(* CODESYS project lcls-twincat-motion-v4.0.8.library
   Title: lcls-twincat-motion
   Version: 4.0.8
   Placeholder: lcls-twincat-motion
   Company: SLAC

Project tree, tasks and I/O mapping:
  libraries: LCLS General, * (SLAC); PMPS, * (SLAC - LCLS); Tc2_EtherCAT, * (Beckhoff Automation GmbH); Tc2_Math, * (Beckhoff Automation GmbH); Tc2_MC2, * (Beckhoff Automation GmbH); Tc2_Standard, * (Beckhoff Automation GmbH); Tc2_System, * (Beckhoff Automation GmbH); Tc2_Utilities, * (Beckhoff Automation GmbH); Tc3_JsonXml, * (Beckhoff Automation GmbH); Tc3_Module, * (Beckhoff Automation GmbH); TcUnit, * (www.tcunit.org)
  DUTs/
    Deprecated/
      data type DUT_MotionPneumaticActuator
      data type DUT_MotionStage
      data type DUT_PositionState
      data type EL5042_Status
      data type ENUM_EpicsHomeCmd
      data type ENUM_EpicsInOut
      data type ENUM_EpicsInOut_INT
      data type ENUM_EpicsMotorCmd
      data type ENUM_MotionFFType
      data type ENUM_MotionRequest
      data type ENUM_PnuematicActuatorPositionState
      data type ENUM_StageBrakeMode
      data type ENUM_StageEnableMode
      data type ENUM_StatePMPSStatus
    data type E_EpicsHomeCmd
    data type E_EpicsInOut
    data type E_EpicsMotorCmd
    data type E_LCLSMotionError
    data type E_MotionFFType
    data type E_MotionRequest
    data type E_PnuematicActuatorPositionState
    data type E_StageBrakeMode
    data type E_StageEnableMode
    data type E_StatePMPSStatus
    data type ST_AxisParameterSetExposed
    data type ST_EL5042_Status
    data type ST_MotionPneumaticActuator
    data type ST_MotionStage
    data type ST_PositionState
    data type ST_RenishawAbsEnc
    data type ST_StateEpicsToPlc
    data type ST_StatePlcToEpics
    data type ST_StatePMPSEpicsToPlc
    data type ST_StatePMPSPlcToEpics
  GVLs/
    global variables MOTION_GVL
    global variables MotionConstants
  POUs/
    Deprecated/
      function block FB_EpicsInOut [ST]
      function block FB_PositionStateBase [ST]: Exec, StateHandler
      function block FB_PositionStateBase_WithPMPS [ST]: Exec, PMPSHandler
      function block FB_PositionStateBase_WithPMPS_Test [ST]: Exec, PMPSHandler
      function block FB_PositionStateInOut [ST]
      function block FB_PositionStateInOut_WithPMPS [ST]
      function block FB_PositionStateInOut_WithPMPS_Test [ST]
      function block FB_PositionStateManager [ST]
      function block FB_PositionStatePMPS [ST]: AssertHere, ClearAsserts, HandleBPTM, HandleFFO, HandlePmpsDb
      function block FB_PositionStatePMPS_Base [ST]: AssertHere, ClearAsserts, Exec, GetBeamFromState, GetStateCode, GetStateStruct, HandleBPTM, HandleFFO, HandlePmpsDb
      function block FB_PositionStatePMPS_Test [ST]: HandleBPTM, HandleFFO
      function block FB_StatePTPMove [ST]
    ImplicitChecks/
      function CheckBounds [ST]
      function CheckDivDInt [ST]
      function CheckDivLInt [ST]
      function CheckDivLReal [ST]
      function CheckDivReal [ST]
    Motion/
      Gantry/
        function block FB_GantryAutoCoupling [ST]
        function block FB_GantryDiffVirtualLimitSwitch [ST]
      PMPS/
        function block FB_EncErrorFFO [ST]
        function block FB_MiscStatesErrorFFO [ST]
        function block FB_MotionBPTM [ST]: CheckCount, HandleTimeout, RunBPTM, SetDoneMoving
        function block FB_MotionClearAsserts [ST]
        function block FB_MotionReadPMPSDBND [ST]: BackfillInfo, ReadDatabase, RunFastFaults, SelectLookupKeys
        function block FB_NCErrorFFO [ST]
        function block FB_PerMotorFFOND [ST]: CheckCount, HandleFFO, HandleLoops
        function block FB_PositionStatePMPS1D [ST]
        function block FB_PositionStatePMPS2D [ST]
        function block FB_PositionStatePMPS3D [ST]
        function block FB_PositionStatePMPSND_Core [ST]
        function block FB_Standard_PMPSDB [ST]
        function block FB_StatePMPSEnables [ST]: ApplyEnables, GetBounds, RunFastFaults, SetEnables
        function block FB_StatePMPSEnablesND [ST]: CheckCount, DoLimits, RunFastFaults
      States/
        Examples/
          function block FB_PositionState1D_InOut [ST]
          function block FB_PositionState2D_InOut [ST]
          function block FB_PositionStatePMPS1D_InOut [ST]
          function block FB_PositionStatePMPS2D_InOut [ST]
        Helpers/
          function F_AtPositionState [ST]
          function F_PosOverLowerBound [ST]
          function F_PosUnderUpperBound [ST]
          function F_PosWithinDelta [ST]
          function block FB_RawCountConverter [ST]
        Internals/
          function block FB_PositionStateInternal [ST]
          function block FB_PositionStateInternalND [ST]
          function block FB_PositionStateLock [ST]
        function block FB_PositionState1D [ST]
        function block FB_PositionState2D [ST]
        function block FB_PositionState3D [ST]
        function block FB_PositionStateMove [ST]
        function block FB_PositionStateMoveND [ST]: CheckCount, CombineOutputs, DoStateMoves
        function block FB_PositionStateND_Core [ST]
        function block FB_PositionStateRead [ST]
        function block FB_PositionStateReadND [ST]: CheckCount, CombineOutputs, DoStateReads
        function block FB_StateSetupHelper [ST]
        function block FB_StatesInputHandler [ST]
      Utils/
        function F_MotionErrorCodeLookup [ST]
        function block FB_SetEnables [ST]
      function block FB_EncoderValue [ST]
      function block FB_EncSaveRestore [ST]
      function block FB_LogMotionError [ST]
      function block FB_MotionHoming [ST]
      function block FB_MotionPneumaticActuator [ST]: ACT_IO, ACT_Logger
      function block FB_MotionRequest [ST]
      function block FB_MotionStage [ST]
      function block FB_MotionStageNCParams [ST]
      function block FB_MotionStageSim [ST]
    MotorTesting/
      function block FB_MicroStepCountTest [ST]
  tc_mca_std_lib/
    DUTs/
      data type DUT_AxisStatus_v0_01
    GVLs/
      global variables GVL
    POUs/
      ChangeConfig/
        function block FB_ReadFloatParameter [ST]
        function block FB_ReadParameterInNc_v1_00 [ST]
        function block FB_WriteFloatParameter [ST]
        function block FB_WriteParameterInNc_v1_00 [ST]
      ErrorHandling/
        data type DUT_ErrorState
        data type DUT_TerminalError
        function block FB_ErrorList [ST]
        function block FB_TerminalError [ST]
        global variables GVL_ErrorSystem
        data type ST_ErrorSystem
      Hardware/
        EtherCAT_Terminals/
          Analog_Inputs/
            function block EL3174_0002 [ST]
            function block EL3214 [ST]
            function block EL3255 [ST]
            function block FB_CalculateFrequency_3702_v0_01 [ST]
          Digital_Inputs/
            function block EL1008 [ST]
            function block EL1018 [ST]
            function block EL1808 [ST]
            function block EL1809 [ST]
            function block EL1819 [ST]
            function block FB_EL1252ASM_v1_00 [ST]
          Digital_Outputs/
            External_Types/
              data type dutEL2521_Ctrl
              data type dutEL2521_Status
            function block EL2014 [ST]
            function block EL2252 [ST]
            function block EL2808 [ST]
            function block EL2819 [ST]
          Measuring_Terminals/
            function block EL5002 [ST]
            function block EL5021 [ST]
            function block EL5042 [ST]
            function block EL5101 [ST]
          Motion/
            function block EL7211_v1_00 [ST]
            function block EL9576_v1_00 [ST]
          System/
            function block EL9410 [ST]
            function block EL9505 [ST]
        Other/
          function block EK1200 [ST]
      Motion/
        Homing/
          function block FB_HomeDirect [ST]
          function block FB_HomeFinish [ST]
          function block FB_HomePrepare [ST]
          function block FB_HomeReadNcVelocities [ST]
          function block FB_HomeReadSoftLimEnable [ST]
          function block FB_HomeToSwitch [ST]
          function block FB_HomeVirtual [ST]
          function block FB_HomeWriteNcVelocities [ST]
          function block FB_HomeWriteSoftLimEnable [ST]
        function block FB_DriveVirtual [ST]
        function block FB_NcAxis [ST]
  Tests/
    Helpers/
      data type E_TestStates
      function block FB_CauseNCError [ST]
      function block FB_MotorTestSuite [ST]: SetEnables, SetEnablesPMPS, SetGoodState
      function block FB_PMPSJsonTestHelper [ST]: bitmaskToString
      function block FB_TestHelperSetAndMove [ST]
    function block FB_AtPositionState_Test [ST]: TestAtPositionStateInvalid, TestAtPositionStateJustRight, TestAtPositionStateLeave, TestAtPositionStateTooHigh, TestAtPositionStateTooLow, TestAtPositionStateTweak, TestAtPositionStateWithoutInternal, TestPosOverLowerBoundNo, TestPosOverLowerBoundYes, TestPosUnderUpperBoundNo, TestPosUnderUpperBoundYes, TestPosWithinDeltaJustRight, TestPosWithinDeltaTooHigh, TestPosWithinDeltaTooLow
    function block FB_AxisParameterSetExposed_Test [ST]: TestParameterCopy
    function block FB_MiscStatesErrorFFO_Test [ST]: TestBeamParamsNotOk, TestDebounce, TestTransitionState, TestUnknownState, TestZeroRate, TripUntrip
    function block FB_MotionBPTM_Test [ST]: AssertInPool, SetMotorDone, SetMotorMoving, SetMotorStartup, Test3dMove, TestCount, TestInit, TestNoMove
    function block FB_MotionClearAsserts_Test [ST]: TestBasic
    function block FB_MotionReadPMPSDBND_Test [ST]: TestBackfill, TestDupe, TestHalfFull, TestNonsense, TestSolo, TestTrio
    function block FB_NCErrorFFO_Test [ST]: TestEnc, TestNC
    function block FB_PerMotorFFOND_Test [ST]: TestBlankCount, TestTwoMotorEncError
    function block FB_PositionStateMove_Test [ST]: TestBadStates, TestMove, TestMoveOk
    function block FB_PositionStateMoveND_Test [ST]: ResetGoals, TestMove
    function block FB_PositionStateND_Test [ST]: Test1D, Test2D, Test3D, TestInputDeadlock
    function block FB_PositionStatePMPSND_Test [ST]: AssertMotionLims, Test1D, Test2D, Test3D, TestStartup1D, TestStartup2D, TestStartup3D
    function block FB_PositionStateRead_Test [ST]: Asserts, TestDupe, TestMovingPosition, TestStaticPosition
    function block FB_PositionStateReadND_Test [ST]: DoAssert, DoMove, DoRead, PerMotor, SquareSetup, TestCombos, TestForgot, TestSquare
    function block FB_StatePMPSEnables_Test [ST]: TestAbove, TestAt, TestBelow, TestDisabled, TestInvalid, TestLimits, TestMoveAt, TestMoveTo, TestNotUpdated
    function block FB_StatePMPSEnablesND_Test [ST]: TestCount, TestMaint, TestUnderOverGoals
    function block FB_StateSetupHelper_Test [ST]: TestDefaultOnly, TestManyOverrides, TestNoDefault, TestNormalCase, TestOnlyOnce
    function block FB_TestHelperSetAndMove_Test [ST]: BasicMotion
    function block FB_TestStateInitTiming [ST]: PassiveReinit
    program PRG_TEST [ST]
  Version/
    global variables Global_Version
*)

// DUTs/Deprecated/DUT_MotionPneumaticActuator
{attribute 'obsolete' := 'DUT_MotionPneumaticActuator has been renamed to ST_MotionPneumaticActuator'}
TYPE DUT_MotionPneumaticActuator : ST_MotionPneumaticActuator; END_TYPE

// DUTs/Deprecated/DUT_MotionStage
{attribute 'obsolete' := 'DUT_MotionStage has been renamed to ST_MotionStage'}
TYPE DUT_MotionStage : ST_MotionStage; END_TYPE

// DUTs/Deprecated/DUT_PositionState
{attribute 'obsolete' := 'DUT_PositionState has been renamed to ST_PositionState'}
TYPE DUT_PositionState : ST_PositionState; END_TYPE

// DUTs/Deprecated/EL5042_Status
{attribute 'obsolete' := 'EL5042_Status has been renamed to ST_EL5042_Status'}
TYPE EL5042_Status : ST_EL5042_Status; END_TYPE

// DUTs/Deprecated/ENUM_EpicsHomeCmd
{attribute 'obsolete' := 'Use E_EpicsHomeCmd'}
TYPE ENUM_EpicsHomeCmd : E_EpicsHomeCmd; END_TYPE

// DUTs/Deprecated/ENUM_EpicsInOut
{attribute 'obsolete' := 'Use E_EpicsInOut'}
TYPE ENUM_EpicsInOut : E_EpicsInOut; END_TYPE

// DUTs/Deprecated/ENUM_EpicsInOut_INT
{attribute 'obsolete' := 'Use ENUM_EpicsInOut'}
{attribute 'qualified_only'}
// Example EPICS states enum for use in all versions of the states FBs
// Remove strict attribute for easier handling
TYPE ENUM_EpicsInOut_INT :
(
    UNKNOWN := 0, // UNKNOWN must be in slot 0 or the FB breaks
    OUT := 1, // OUT at slot 1 is a convention
    IN := 2
) INT;
END_TYPE

// DUTs/Deprecated/ENUM_EpicsMotorCmd
{attribute 'obsolete' := 'Use E_EpicsMotorCmd'}
TYPE ENUM_EpicsMotorCmd : E_EpicsMotorCmd; END_TYPE

// DUTs/Deprecated/ENUM_MotionFFType
{attribute 'obsolete' := 'Use E_MotionFFType'}
TYPE ENUM_MotionFFType : E_MotionFFType; END_TYPE

// DUTs/Deprecated/ENUM_MotionRequest
{attribute 'obsolete' := 'Use E_MotionRequest'}
TYPE ENUM_MotionRequest : E_MotionRequest; END_TYPE

// DUTs/Deprecated/ENUM_PnuematicActuatorPositionState
{attribute 'obsolete' := 'Use E_PnuematicActuatorPositionState'}
TYPE ENUM_PnuematicActuatorPositionState : E_PnuematicActuatorPositionState; END_TYPE

// DUTs/Deprecated/ENUM_StageBrakeMode
{attribute 'obsolete' := 'Use E_StageBrakeMode'}
TYPE ENUM_StageBrakeMode : E_StageBrakeMode; END_TYPE

// DUTs/Deprecated/ENUM_StageEnableMode
{attribute 'obsolete' := 'Use E_StageEnableMode'}
TYPE ENUM_StageEnableMode : E_StageEnableMode; END_TYPE

// DUTs/Deprecated/ENUM_StatePMPSStatus
{attribute 'obsolete' := 'Use E_StatePMPSStatus'}
TYPE ENUM_StatePMPSStatus : E_StatePMPSStatus; END_TYPE

// DUTs/E_EpicsHomeCmd
{attribute 'qualified_only'}
{attribute 'strict'}
TYPE E_EpicsHomeCmd :
    // Defines the valid options for homing in FB_MotionStage
(
    LOW_LIMIT := 1, // Low limit switch
    HIGH_LIMIT := 2, // High limit switch
    HOME_VIA_LOW := 3, // Home switch via low switch
    HOME_VIA_HIGH := 4, // Home switch via high switch
    ABSOLUTE_SET := 15, // Set here to be fHomePosition
    NONE := -1 // Do not home, ever
);
END_TYPE

// DUTs/E_EpicsInOut
{attribute 'qualified_only'}
// Example EPICS states enum for use in all versions of the states FBs
// Remove strict attribute for easier handling
TYPE E_EpicsInOut :
(
    UNKNOWN := 0, // UNKNOWN must be in slot 0 or the FB breaks
    OUT := 1, // OUT at slot 1 is a convention
    IN := 2
) UINT;
END_TYPE

// DUTs/E_EpicsMotorCmd
{attribute 'qualified_only'}
{attribute 'strict'}
TYPE E_EpicsMotorCmd :
    // Defines valid EPICS commands for nCommand
(
    JOG := 0,
    MOVE_VELOCITY := 1,
    MOVE_RELATIVE := 2,
    MOVE_ABSOLUTE := 3,
    MOVE_MODULO := 4,
    HOME := 10,
    GEAR := 30
);
END_TYPE

// DUTs/E_LCLSMotionError
{attribute 'qualified_only'}
{attribute 'strict'}
TYPE E_LCLSMotionError :
(
    ABORTED := 16#7900,
    UNSAFE := 16#7901,
    INVALID := 16#7902,
    TEST := 16#FFFF
) UDINT;
END_TYPE

// DUTs/E_MotionFFType
{attribute 'qualified_only'}
TYPE E_MotionFFType :
(
    STOPPER_FAULT := 16#1000,
    ZERO_RATE := 16#1001,
    BPTM_TIMEOUT := 16#1002,
    BPTM_ERROR := 16#1003,
    MAINT_MODE := 16#1004,
    NOT_A_STATE := 16#1005,
    INVALID_GOAL := 16#1006,
    TOO_MANY_TRIPS := 16#1007,
    BP_MISMATCH := 16#1008,
    INTERNAL_ERROR := 16#1009,
    PNEUMATIC_MOVE := 16#1010,
    MOT_GENERIC := 16#1011,
    LOW_RESERVED_NC := 16#2000,
    HIGH_RESERVED_NC := 16#20FF,
    DEVICE_MOVE := 16#2100
) UINT := MOT_GENERIC;
END_TYPE

// DUTs/E_MotionRequest
{attribute 'qualified_only'}
{attribute 'strict'}
TYPE E_MotionRequest :
    // Defines behavior options for when FB_MotionRequest is run during an active move from another source
(
    WAIT := 0,
    INTERRUPT := 1,
    ABORT := 2
);
END_TYPE

// DUTs/E_PnuematicActuatorPositionState
{attribute 'qualified_only'}
{attribute 'strict'}
// Defines the positions for a pnuematic actuator
TYPE E_PnuematicActuatorPositionState :
(
   RETRACTED    := 0, // Out limit switch is active
   INSERTED    := 1, // In limit switch is active
   MOVING    := 2, // Neither limit switches is Active
   INVALID :=3 // Invalid state
);
END_TYPE

// DUTs/E_StageBrakeMode
{attribute 'qualified_only'}
{attribute 'strict'}
TYPE E_StageBrakeMode :
    // Defines when to send the brake disengage signal in FB_MotionStage
(
    IF_ENABLED, // Disengage brake when the motor is enabled
    IF_MOVING, // Disengage brake when the motor is moving
    NO_BRAKE // Do not change the brake state in FB_MotionStage
);
END_TYPE

// DUTs/E_StageEnableMode
{attribute 'qualified_only'}
{attribute 'strict'}
TYPE E_StageEnableMode :
    // Define conditions when FB_MotionStage automatically sets bEnable
(
    ALWAYS, // Always set bEnable to TRUE
    NEVER,  // Only change bEnable on errors
    DURING_MOTION  // Enable before motion, disable after motion
);
END_TYPE

// DUTs/E_StatePMPSStatus
{attribute 'qualified_only'}
{attribute 'strict'}
TYPE E_StatePMPSStatus :
(
    // No other enum state describes it
    UNKNOWN := 0,
    // Moving toward a known state
    TRANSITION := 1,
    // Within a known state, not trying to leave
    AT_STATE := 2,
    // PMPS is in some way disabled, either with maint mode or arbiter disable
    DISABLED := 3
);
END_TYPE

// DUTs/ST_AxisParameterSetExposed
TYPE ST_AxisParameterSetExposed :
    // Collects the axis parameters that are intentionally exposed to EPICS.
STRUCT
    // Maximum Dynamics
    {attribute 'pytmc' := '
        pv: MaxVel
        io: i
        field: DESC Maximum commandable speed of the axis in EU/s.
    '}
    fVeloMaximum                : LREAL; // Maximum commandable speed of the axis in EU/s.
    {attribute 'pytmc' := '
        pv: MaxAccel
        io: i
        field: DESC Maximum rate of increase in speed of the axis in EU/s^2.
    '}
    fAccelerationMax            : LREAL; // Maximum rate of increase in speed of the axis in EU/s^2.
    {attribute 'pytmc' := '
        pv: MaxDecel
        io: i
        field: DESC Maximum rate of decrease in speed of the axis in EU/s^2.
    '}
    fDecelerationMax            : LREAL; // Maximum rate of decrease in speed of the axis in EU/s^2.

    // Monitoring
    {attribute 'pytmc' := '
        pv: PosLagEn
        io: i
        field: DESC TRUE if position lag monitor (also known as stall monitor) is enabled.
    '}
    bCtrlEnablePosDiffControl   : WORD;  // Enable/Disable state of Position Lag Monitor.
    {attribute 'pytmc' := '
        pv: PosLagVal
        io: i
        field: DESC Maximum magnitude of position lag in EU.
    '}
    fCtrlPosDiffMax             : LREAL; // Maximum magnitude of position lag in EU.
    {attribute 'pytmc' := '
        pv: PosLagTime
        io: i
        field: DESC Maximum allowable duration outside of maximum position lag value in seconds.
    '}
    fCtrlPosDiffMaxTime         : LREAL; // Maximum allowable duration outside of maximum position lag value in seconds.

    // Limit Switches
    {attribute 'pytmc' := '
        pv: SLimMinEn
        io: i
        field: DESC TRUE if controller static minimum limit is enabled.
    '}
    bEncEnableSoftEndMinControl : WORD;  // Enable/Disable state of controller static minimum limit.
    {attribute 'pytmc' := '
        pv: SLimMaxEn
        io: i
        field: DESC TRUE if controller static maximum limit is enabled.
    '}
    bEncEnableSoftEndMaxControl : WORD;  // Enable/Disable state of controller static maximum limit.
    {attribute 'pytmc' := '
        pv: SLimMin
        io: i
        field: DESC Minimum commandable position of the axis in EU.
    '}
    fEncSoftEndMin              : LREAL; // Minimum commandable position of the axis in EU.
    {attribute 'pytmc' := '
        pv: SLimMax
        io: i
        field: DESC Maximum commandable position of the axis in EU.
    '}
    fEncSoftEndMax              : LREAL; // Maximum commandable position of the axis in EU.

    // Encoder Evaluation
    {attribute 'pytmc' := '
        pv: EncScaling
        io: i
        field: DESC Encoder scaling numerator / denominator in EU/COUNT.
    '}
    fEncScaleFactorInternal      : LREAL; // Encoder scaling numerator / denominator in EU/COUNT.
    {attribute 'pytmc' := '
        pv: EncOffset
        io: i
        field: DESC Encoder offset in EU.
    '}
    fEncOffset                   : LREAL; // Encoder offset in EU.

END_STRUCT
END_TYPE

// DUTs/ST_EL5042_Status
TYPE ST_EL5042_Status :
STRUCT
END_STRUCT
END_TYPE

// DUTs/ST_MotionPneumaticActuator
{attribute 'qualified_only'}
{attribute 'strict'}
TYPE ST_MotionPneumaticActuator :
    // Defines the EPICS interface to actuating a pneumatic stage
STRUCT
     (* Hardware *)
    //Readbacks
    //Limit Switch
    {attribute 'pytmc' := '
     pv: PLC:bInLimitSwitch
     io: i
     field: ZNAM FALSE
     field: ONAM TRUE
     field: DESC TRUE if IN limit is reached
    '}
    i_bInLimitSwitch    :    BOOL;
    {attribute 'pytmc' := '
     pv: PLC:bOutLimitSwitch
     io: i
     field: ZNAM FALSE
     field: ONAM TRUE
     field: DESC TRUE if OUT limit is reached
    '}
    i_bOutLimitSwitch    :    BOOL;
    //Controls
    //Digital outputs
    {attribute 'pytmc' := '
    pv: bRetractDigitalOutput;
    io: i;
    field: ONAM FALSE
    field: ZNAM TRUE
    field: DESC TRUE if Retract digital output is active
    '}
    q_bRetract    :    BOOL;
    {attribute 'pytmc' := '
    pv: bInsertDigitalOutput;
    io: i;
    field: ONAM FALSE
    field: ZNAM TRUE
    field: DESC TRUE if Insert digital output is active
    '}
    q_bInsert    :    BOOL;


    //Logic and supervisory
    {attribute 'pytmc' := '
    pv: bInterlockOK;
    io: i;
    field: ZNAM FALSE
    field: ONAM TRUE
    field: DESC True if the actuator has permission to move in either direction
    '}
    bILK_OK: BOOL;
    {attribute 'pytmc' := '
    pv: bInsertEnable;
    io: i;
    field: ZNAM FALSE
    field: ONAM TRUE
    field: DESC True if the actuator had permission to be retracted
    '}
    bInsertOK    :    BOOL;
    {attribute 'pytmc' := '
    pv: bRetractEnable;
    io: i;
    field: ZNAM FALSE
    field: ONAM TRUE
    field: DESC True if the actuator had permission to be inserted
    '}
    bRetractOK    :    BOOL;

    (* Commands *)
    // Used from Epics to comand the actuator to  move
    {attribute 'pytmc' := '
    pv: CMD:IN;
    io: io;
    field: DESC Used by EPICS and internally to request Insert motion
    '}
    bInsert_SW        :    BOOL;
    {attribute 'pytmc' := '
    pv: CMD:OUT;
    io: io;
    field: DESC Used by EPICS and internally to request retract motion
    '}
    bRetract_SW    :    BOOL;

    (*Returns*)
     // TRUE if in the middle of a command
    {attribute 'pytmc' := '
     pv: bBusy
     io: i
     field: ONAM FALSE
     field: ZNAM TRUE
     field: DESC TRUE if in the middle of a command
    '}
    bBusy: BOOL;
    // TRUE if we've done a command and it has finished
    {attribute 'pytmc' := '
     pv: bDone
     io: i
     field: ONAM FALSE
     field: ZNAM TRUE
      field: DESC TRUE if command finished successfully
    '}
    bDone: BOOL;
     {attribute 'pytmc' := '
        pv: bReset
        io: io
        field: ZNAM FALSE
        field: ONAM TRUE
        field: DESC Used internally to reset errors
    '}
    bReset: BOOL;
    // TRUE if we're in an error state
    {attribute 'pytmc' := '
     pv: PLC:bError
     io: i
     field: ONAM FALSE
     field: ZNAM TRUE
     field: DESC TRUE if we're in an error state
    '}
    bError: BOOL;

     // Error code if nonzero
    {attribute 'pytmc' := '
     pv: PLC:nErrorId
     io: i
     field: DESC Error code if nonzero
    '}
    nErrorId: UDINT;
    // Message to identify the error state
    {attribute 'pytmc' := '
     pv: PLC:sErrorMessage
     io: i
     field: DESC Message to identify the error state
    '}
    sErrorMessage: STRING;
    {attribute 'pytmc' := '
    pv: nPositionState ;
    type: mbbi ;
    field: ZRST RETRACTED ;
    field: ONST INSERTED ;
    field: TWST MOVING ;
    field: THST INVALID ;
    io: i
    field: DESC Pneumatic actuator position
    '}

    eState    :    E_PnuematicActuatorPositionState := E_PnuematicActuatorPositionState.INVALID;

END_STRUCT
END_TYPE

// DUTs/ST_MotionStage
TYPE ST_MotionStage :
    // Defines the EPICS interface to moving a motor in TwinCAT
STRUCT
    (* Hardware *)

    // PLC Axis Reference
    Axis: AXIS_REF;
    // NC Forward Limit Switch: TRUE if ok to move
    bLimitForwardEnable AT %I*: BOOL;
    // NC Backward Limit Switch: TRUE if ok to move
    bLimitBackwardEnable AT %I*: BOOL;
    // NO Home Switch: TRUE if at home
    bHome AT %I*: BOOL;
    // NC Brake Output: TRUE to release brake
    bBrakeRelease AT %Q*: BOOL;
    // NC STO Input: TRUE if ok to move
    {attribute 'pytmc' := '
        pv: PLC:bHardwareEnable
        io: i
        field: ZNAM FALSE
        field: ONAM TRUE
        field: DESC TRUE if STO not hit
    '}
    bHardwareEnable AT %I*: BOOL;

    // Raw encoder IO for ULINT (Biss-C)
    nRawEncoderULINT AT %I*: ULINT;
    // Raw encoder IO for UINT (Relative Encoders)
    nRawEncoderUINT AT %I*: UINT;
    // Raw encoder IO for INT (LVDT)
    nRawEncoderINT AT %I*: INT;

    (* Psuedo-hardware *)

    // Forward enable EPS summary
    bAllForwardEnable: BOOL:=FALSE;
    // Backward enable EPS summary
    bAllBackwardEnable: BOOL:=FALSE;
    // Enable EPS summary encapsulating emergency stop button and any additional motion preventive hardware
    bAllEnable: BOOL:=FALSE;
    // Forward virtual gantry limit switch
    bGantryForwardEnable: BOOL:=FALSE;
    // Backward virtual gantry limit switch
    bGantryBackwardEnable: BOOL:=FALSE;
    // Encoder count summary, if linked above
    {attribute 'pytmc' := '
        pv: PLC:nEncoderCount
        io: i
        field: DESC Count from encoder hardware
    '}
    nEncoderCount: UDINT;
    // Forward Enable EPS struct
    {attribute 'pytmc' := '
        pv: PLC:stEPSF
        io: i
        field: DESC Forward Enable Interlocks
    '}
    stEPSForwardEnable: DUT_EPS;
    // Backward Enable EPS struct
    {attribute 'pytmc' := '
        pv: PLC:stEPSB
        io: i
        field: DESC Backward Enable Interlocks
    '}
    stEPSBackwardEnable: DUT_EPS;
    // Power Enable EPS struct
    {attribute 'pytmc' := '
        pv: PLC:stEPSP
        io: i
        field: DESC Power Interlocks
    '}
    stEPSPowerEnable: DUT_EPS;

    (* Settings *)
    // Name to use for log messages, fast faults, etc.
    sName: STRING;
    // If TRUE, we want to enable the motor independently of PMPS or other safety systems.
    bPowerSelf: BOOL:=FALSE;
    // Determines when we automatically enable the motor
    nEnableMode: E_StageEnableMode:=E_StageEnableMode.DURING_MOTION;
    // Determines when we automatically disengage the brake
    nBrakeMode: E_StageBrakeMode:=E_StageBrakeMode.IF_ENABLED;
    // Determines our encoder homing strategy
    nHomingMode: E_EpicsHomeCmd:=E_EpicsHomeCmd.NONE;
    // Set true to activate gantry EPS
    bGantryAxis: BOOL:=FALSE;

    // Set to gantry difference tolerance
    nGantryTol: LINT:=0;

    // Encoder count at which this axis is aligned with other axis
    nEncRef: ULINT:=0;

    (* Commands *)
    // Used internally to request enables
    bEnable: BOOL;
    // Used internally to reset errors and other state
    {attribute 'pytmc' := '
        pv: PLC:bReset
        io: io
        field: ZNAM FALSE
        field: ONAM TRUE
        field: DESC Used internally to reset errors
    '}
    bReset: BOOL;
    // Used internally and by the IOC to start or stop a move
    bExecute: BOOL;
    // Used by the IOC to disable an axis
    {attribute 'pytmc' := '
        pv: PLC:bUserEnable
        io: io
        field: ZNAM DISABLE
        field: ONAM ENABLE
        field: DESC Used to disable power entirely for an axis
    '}
    bUserEnable: BOOL := 1;

    (* Shortcut Commands *)
    // Start a move to fPosition with fVelocity
    bMoveCmd: BOOL;
    // Start the homing routine
    {attribute 'pytmc' := '
        pv: PLC:bHomeCmd
        io: io
        field: DESC Start the homing routine
    '}
    bHomeCmd: BOOL;

    (* Command Args *)
    // Used internally and by the IOC to pick what kind of move to do
    nCommand: INT;
    // Used internally and by the IOC to pass additional data to some commands
    nCmdData: INT;
    // Used internally and by the IOC to pick a destination for the move
    fPosition: LREAL;
    // Used internally and by the IOC to pick a move velocity
    fVelocity: LREAL;
    // Used internally and by the IOC to pick a move acceleration
    fAcceleration: LREAL;
    // Used internally and by the IOC to pick a move deceleration
    fDeceleration: LREAL;
    // Used internally and by the IOC to pick a home position
    {attribute 'pytmc' := '
        pv: PLC:fHomePosition
        io: io
        field: DESC Used internally and by the IOC to pick home position
    '}
    fHomePosition: LREAL;

    (* Info *)
    // Unique ID assigned to each axis in the NC
    nMotionAxisID: UDINT:=0;

    (* Returns *)
    // TRUE if done enabling
    bEnableDone: BOOL;
    // TRUE if in the middle of a command
    bBusy: BOOL;
    // TRUE if we've done a command and it has finished
    bDone: BOOL;
    // TRUE if the motor has been homed, or does not need to be homed
    bHomed: BOOL;
    // TRUE if we have safety permission to move
    bSafetyReady: BOOL;
    // TRUE if we're in an error state
    {attribute 'pytmc' := '
        pv: PLC:bError
        io: i
        field: ZNAM FALSE
        field: ONAM TRUE
        field: DESC TRUE if we are in an error state
        update: 100Hz notify
    '}
    bError: BOOL;
    // Error code if nonzero
    {attribute 'pytmc' := '
        pv: PLC:nErrorId
        io: i
        field: DESC Error code if nonzero
        update: 100Hz notify
    '}
    nErrorId: UDINT;
    // Message to identify the error state
    {attribute 'pytmc' := '
        pv: PLC:sErrorMessage
        io: i
        field: DESC Message to identify the error state
        update: 100Hz notify
    '}
    sErrorMessage: STRING;
    // Internal hook for custom error messages
    sCustomErrorMessage: STRING;
    // MC_ReadParameterSet Output
    stAxisParameters: ST_AxisParameterSet;
    // NC parameters that are exposed with pytmc pragmas
    {attribute 'pytmc' := '
        pv: PLC:AxisPar
        io: i
        field: DESC Axis configuration parameters in the numerical controller.
    '}
    stAxisParametersExposed: ST_AxisParameterSetExposed;
    // True if we've updated stAxisParameters at least once
    bAxisParamsInit: BOOL;

    // Misc axis status information for the IOC
    stAxisStatus: DUT_AxisStatus_v0_01;

    (* Other status information for users of the IOC *)
    // Position lag difference
    {attribute 'pytmc' := '
        pv: PLC:fPosDiff
        io: i
        field: DESC Position lag difference
    '}
    fPosDiff: LREAL;
END_STRUCT
END_TYPE

// DUTs/ST_PositionState
TYPE ST_PositionState :
    // Defines settings and current safety status for moves to specific positions for an axis
STRUCT
    // Name as queried via the NAME PV in EPICS
    {attribute 'pytmc' := '
        pv: NAME
        io: input
        field: DESC Name of this position state
    '}
    sName: STRING := 'Invalid';

    // Position associated with this state
    {attribute 'pytmc' := '
        pv: SETPOINT
        io: io
        field: DESC Axis position associated with this state
    '}
    fPosition: LREAL;

    {attribute 'pytmc' := '
        pv: ENCODER
        io: i
        field: DESC Encoder count associated with this state
    '}
    nEncoderCount: UDINT;

    // Maximum allowable deviation from fPosition while at the state
    fDelta: LREAL;

    // Speed at which to move to this state
    {attribute 'pytmc' := '
        pv: VELO
        io: io
        field: DESC Speed at which to move to this state
    '}
    fVelocity: LREAL;

    // (optional) Acceleration to use for moves to this state
    fAccel: LREAL;

    // (optional) Deceleration to use for moves to this state
    fDecel: LREAL;

    // Safety parameter. This must be set to TRUE by the PLC program to allow moves to this state. This is expected to change as conditions change.
    {attribute 'pytmc' := '
        pv: MOVE_OK
        io: i
        field: ZNAM FALSE
        field: ONAM TRUE
        field: DESC TRUE if the move would be safe
    '}
    bMoveOk: BOOL;

    // Signifies to FB_PositionStateLock that this state should be immutable
    bLocked: BOOL;

    // Set this to TRUE when you make your state. This defaults to FALSE so that uninitialized states can never be moved to
    bValid: BOOL;

    // Set this to TRUE when you want to use the raw encoder counts to define the state
    bUseRawCounts: BOOL;

    // Is set to TRUE by FB_PositionStateInternal when called
    bUpdated: BOOL;

    // We give this a state name and it is used to load parameters from the pmps database.
    stPMPS: ST_DbStateParams;
END_STRUCT
END_TYPE

// DUTs/ST_RenishawAbsEnc
// Renishaw BiSS-C absolute encoder used with an EL5042
TYPE ST_RenishawAbsEnc :
STRUCT
    Count AT %I*: ULINT; // Connect to encoder "Position" input
    Status: ST_EL5042_Status; // Status struct placeholder
    Ref: ULINT; // Encoder zero position (useful for aligned position with gantries)
END_STRUCT
END_TYPE

// DUTs/ST_StateEpicsToPlc
TYPE ST_StateEpicsToPlc :
(*
    This data structure contains the standard EPICS input connection points for the state movers.

    The data in this struct flows from EPICS to the PLC.

    It includes everything except the SET PV, which cannot be included here
    as it is sourced from enum values unique to the application, and the PMPS PVs, which are
    gathered in their own data type, ST_StatePMPSEpicsToPlc. That actually means that this only
    holds the RESET PV, for now.

    nSetValue here is actively used by state blocks even though it is not exposed
    directly to EPICS. You should avoid manually modifying it or else
    you may interfere with normal operations of the state function blocks.

    For including your own ENUM input, you should pytmc pragma the PV name to end in "SET",
    and match the prefix of this FB's "RESET" PV. Then, you can include your enum
    as the eEnumSet IN_OUT var and let the EPICS IOC handle it.
*)
STRUCT
    // For internal use only. This holds new goal positions as an integer, else it is 0 if there is no new state move request. It is written to from the user's input enum.
    nSetValue: UINT;

    // Set this to TRUE to acknowledge and clear an error.
    {attribute 'pytmc' := '
        pv: RESET
        io: io
        field: ZNAM False
        field: ONAM True
    '}
    bReset: BOOL;
END_STRUCT
END_TYPE

// DUTs/ST_StatePlcToEpics
TYPE ST_StatePlcToEpics :
(*
    This data structure contains the standard EPICS connection points for the state movers.

    The data in this struct flows from the PLC to EPICS.

    It includes everything except the GET PV, which cannot be included here
    as it is sourced from enum values unique to the application, and the PMPS PVs, which are
    gathered in their own data type, ST_StatePMPSPlcToEpics.

    nGetValue here is actively used by state blocks even though it is not exposed directly
    to EPICS. It is safe to read this value, but you should avoid modifying it, which may
    interfere with normal operations of the state function blocks.

    For including your own ENUM input, you should pytmc pragma the PV name to end in "GET",
    and match the prefix of this FB's "DONE" PV. Then, you can include your enum
    as the eEnumGet IN_OUT var and let the EPICS IOC handle it.
*)
STRUCT
    // For internal use only. This holds the current position index as an integer, else it is 0 if we are changing states or not at any particular state.
    nGetValue: UINT;
    // This will be TRUE when we are in an active state move and FALSE otherwise.
    {attribute 'pytmc' := '
        pv: BUSY
        io: i
        field: ZNAM False
        field: ONAM True
    '}
    bBusy: BOOL;
    // This will be TRUE after a move completes and FALSE otherwise.
    {attribute 'pytmc' := '
        pv: DONE
        io: i
        field: ZNAM False
        field: ONAM True
    '}
    bDone: BOOL;
    // This will be TRUE if the most recent move had an error and FALSE otherwise.
    {attribute 'pytmc' := '
        pv: ERR
        io: i
        field: ZNAM False
        field: ONAM True
    '}
    bError: BOOL;
    // This will be set to an NC error code during an error if one exists or left at 0 otherwise.
    {attribute 'pytmc' := '
        pv: ERRID
        io: i
    '}
    nErrorID: UDINT;
    // This will be set to an appropriate error message during an error if one exists or left as an empty string otherwise.
    {attribute 'pytmc' := '
        pv: ERRMSG
        io: i
    '}
    sErrorMsg: STRING;
END_STRUCT
END_TYPE

// DUTs/ST_StatePMPSEpicsToPlc
TYPE ST_StatePMPSEpicsToPlc :
(*
    This data structure contains the standard PMPS EPICS connection points for the state movers.

    The data in this struct flows from EPICS to the PLC.
*)
STRUCT
    // User setting: TRUE to enable the arbiter, FALSE to disable it.
    {attribute 'pytmc' := '
        pv: PMPS:ARB:ENABLE
        io: io
    '}
    bArbiterEnabled: BOOL := TRUE;
    // User setting: TRUE to enable maintenance mode (Fast fault, free motion), FALSE to disable it.
    {attribute 'pytmc' := '
        pv: PMPS:MAINT
        io: io
    '}
    bMaintMode: BOOL;
END_STRUCT
END_TYPE

// DUTs/ST_StatePMPSPlcToEpics
TYPE ST_StatePMPSPlcToEpics :
(*
    This data structure contains the standard PMPS EPICS connection points for the state movers.

    The data in this struct flows from the PLC to EPICS.
*)
STRUCT
    // The database entry for the transition state. This should always be present.
    {attribute 'pytmc' := '
        pv: PMPS:TRANS
        io: i
    '}
    stTransitionDb: ST_DbStateParams;
END_STRUCT
END_TYPE

// tc_mca_std_lib/DUTs/DUT_AxisStatus_v0_01
TYPE DUT_AxisStatus_v0_01 :
STRUCT
	bEnable: BOOL;
	bReset: BOOL;
	bExecute: BOOL;
	nCommand: UINT;
	nCmdData: UINT;
	fVelocity: LREAL;
	fPosition: LREAL;
	fAcceleration: LREAL;
	fDeceleration: LREAL;
	bJogFwd: BOOL;
	bJogBwd: BOOL;
	bLimitFwd: BOOL;
	bLimitBwd: BOOL;
	fOverride: LREAL := 100;
	bHomeSensor: BOOL;
	bEnabled: BOOL;
	bError: BOOL;
	nErrorId: UDINT;
	fActVelocity: LREAL;
	fActPosition: LREAL;
	fActDiff: LREAL;
	bHomed:BOOL;
	bBusy:BOOL;
END_STRUCT
END_TYPE

// tc_mca_std_lib/POUs/ErrorHandling/DUT_ErrorState
{attribute 'qualified_only'}
{attribute 'strict'}
TYPE DUT_ErrorState :
(
	None,
	Active,
	Inactive,
	Acknowledged
);
END_TYPE

// tc_mca_std_lib/POUs/ErrorHandling/DUT_TerminalError
TYPE DUT_TerminalError :
STRUCT
	//Error system related
	iTerminalID : INT;					//ID of the terminal
	Error_ID : ULINT := 0;				//ID for the Error entry
	ErrorState : DUT_ErrorState;		//State of the error
	
	//Error related
	nDateTimeOn : ULINT;				//Date and time when the error occured. Raw data
	sDateTimeOn : STRING(24);			//Date and time when the error occured. Readable format
	nDateTimeOff : ULINT;				//Date and time when the error disapeared. Raw data
	sDateTimeOff : STRING(24);			//Date and time when the error disapeared. Readable format
	bWcState : BOOL;					//WcState variable of the terminal
	uiInfoDataState : UINT;				//InfoData.State variable of the terminal
	sErrorMessage : STRING (128);		//Error message corresponding to WcState and InfoData.State
	ErrorType : INT; 					//Error types (priorities) need to be developed
END_STRUCT
END_TYPE

// tc_mca_std_lib/POUs/ErrorHandling/ST_ErrorSystem
TYPE ST_ErrorSystem :
STRUCT
	//Array of error data. Size = cSizeOfErrorData in the GVL
	aErrorData : ARRAY [0..GVL_ErrorSystem.cSizeOfErrorData - 1] OF DUT_TerminalError;
	lNextErrorID : ULINT := 1;					//ErrorID for the next error entry
	nNoErrors : UINT;							//Number of errors in the list
	nNoOverflows : INT := 0;					//Number of overflows. How many error entries have been lost
END_STRUCT
END_TYPE

// tc_mca_std_lib/POUs/Hardware/EtherCAT_Terminals/Digital_Outputs/External_Types/dutEL2521_Ctrl
TYPE dutEL2521_Ctrl :
STRUCT
	///The control word (CW) is located in the output process image, and is transmitted from the controller to the terminal.
	///CW.0 FREQ_SEL 0bin / 1bin  Rapid change of the base frequency (only if the ramp function is inactive):
	///0bin = Base frequency 1 (object 8001:02)
	///1bin = Base frequency 2 (object 8001:03) 
	FREQ_SEL: BOOL;
	///CW.1 RAMP_DIS 1bin Operation of the ramp function is cancelled, in spite of object 8000:06 being active; if travel distance control is active, it is interrupted by this bit 
	RAMP_DIS: BOOL;
	///CW.2 GO_COUNTER 1bin  If travel distance control is active (object 8000:0A), then a pre-set counter value is approached when the bit is set 
	GO_COUNTER: BOOL;
	///CW.5 CNT_CLR 1bin The contents of the counter is cleared or set (object 8000:0B) by this bit. 
	///Any overflow or underflow bits that might be set are also cleared by this bit. 
	///The process can be edge triggered or level triggered (object 8000:05). 
	CNT_CLR: BOOL;
END_STRUCT
END_TYPE

// tc_mca_std_lib/POUs/Hardware/EtherCAT_Terminals/Digital_Outputs/External_Types/dutEL2521_Status
TYPE dutEL2521_Status :
STRUCT
	///The status word (SW) is located in the input process image, and is transmitted from the terminal to the controller.
	///SW.0 SEL_ACK/END_COUNTER 1bin  Confirms the change of base frequency. At activated travel distance control: target counter value reached 
	SEL_ACK: BOOL;
	///SW.1 RAMP_ACTIVE 1bin Ramp is currently being followed 
	RAMP_ACTIVE: BOOL;
	///SW.2 UNDERFLOW 1bin This bit is set if the 16-bit counter underflows (0 -> 65535). It is reset when the counter drops below two thirds of its measuring range (43690 -> 43689) or immediately an overflow occurs. 
	UNDERFLOW: BOOL;
	///SW.3 OVERFLOW 1bin This bit is set if the 16-bit counter overflows (65535 -> 0). It is reset when the counter exceeds one third of its measuring range (21845 -> 21846) or immediately an underflow occurs 
	OVERFLOW: BOOL;
	///SW.4 INPUT_T 1bin Status of INPUT_T 
	INPUT_T: BOOL;
	///SW.5 INPUT_Z 1bin Status of INPUT_Z 
	INPUT_Z: BOOL;
	///SW.6 ERROR 1bin General error bit, included with overflow/underflow 
	ERROR: BOOL;
END_STRUCT
END_TYPE

// Tests/Helpers/E_TestStates
{attribute 'qualified_only'}
{attribute 'strict'}
TYPE E_TestStates :
(
    Unknown := 0,
    OUT := 1,
    TARGET1 := 2,
    TARGET2 := 3
) UINT;
END_TYPE

// GVLs/MOTION_GVL
{attribute 'qualified_only'}
VAR_GLOBAL
    // Global file reader instance, used in fbStandardPMPSDB
    fbPmpsFileReader: FB_JsonFileToJsonDoc;
    {attribute 'pytmc' := '
        pv: @(PREFIX)DB
        io: io
    '}
    // Global DB handler, Must be called in PLC project to use the PMPS DB for a motion project
    fbStandardPMPSDB: FB_Standard_PMPSDB;
    // Debug, records the highest number of motors used in an ND states block in the PLC. Can be used to limit MotionConstants.MAX_STATE_MOTORS to save on memory usage and PV count.
    nMaxStateMotorCount: UINT;
    // Debug, records the highest state count in the PLC. Can be used to limit GeneralConstants.MAX_STATES to save on memory usage and PV count.
    nMaxStates: UINT;
END_VAR

// GVLs/MotionConstants
{attribute 'qualified_only'}
(*
    Global Configurable Motion Constants

    These are reconfigurable at the project level.
    When reconfigured they are set prior to compilation and cannot be changed at runtime.
*)
VAR_GLOBAL CONSTANT
    (*
    Arbitary cap on multidimensional states to simplify statements for the compiler.
    This is reconfigurable at the project level and should be set to the highest number of motors used in a states block.
    If you are not sure how many motors are used per state block, check MOTION_GVL.nMaxStateMotorCount
    *)
    MAX_STATE_MOTORS: UINT := 3;
END_VAR

// tc_mca_std_lib/GVLs/GVL
VAR_GLOBAL
	nHomingError:UDINT:=16#14D00;
END_VAR

// tc_mca_std_lib/POUs/ErrorHandling/GVL_ErrorSystem
{attribute 'qualified_only'}
VAR_GLOBAL CONSTANT
	cSizeOfErrorData : UINT := 128;
	
END_VAR

// Version/Global_Version
{attribute 'TcGenerated'}
{attribute 'no-analysis'}
{attribute 'linkalways'}
// This function has been automatically generated from the project information.
VAR_GLOBAL CONSTANT
    {attribute 'const_non_replaced'}
    stLibVersion_lcls_twincat_motion : ST_LibVersion := (iMajor := 4, iMinor := 0, iBuild := 8, iRevision := 0, nFlags := 1, sVersion := '4.0.8');
END_VAR

// POUs/Deprecated/FB_EpicsInOut
{attribute 'obsolete' := 'Use FB_PositionState1D_InOut instead'}
FUNCTION_BLOCK FB_EpicsInOut
// Example usage of FB_PositionStateManager for a simple IN/OUT axis. See NOTE: comments.
// Also usable as a drop-in for these cases (no need to roll your own in/out)
VAR_IN_OUT
    // Motor to apply states to
    stMotionStage: ST_MotionStage;
    // Information about the OUT position
    stOut: ST_PositionState; // NOTE: Do not pragma these, let it happen in the manager.
    // Information about the IN parameter
    stIn: ST_PositionState;
END_VAR
VAR_INPUT
    // If TRUE, the motor will be moved when enumSet is changed
    bEnable: BOOL;
    // When changed, sets the destination and starts a move
    {attribute 'pytmc' := '
        pv: SET
        io: io
    '}
    enumSet: ENUM_EpicsInOut_INT; // NOTE: Please copy this pragma exactly on your enumSet
END_VAR
VAR_OUTPUT
    // If TRUE, we are in an error state
    bError: BOOL; // NOTE: do not pragma these, already has pragma in manager
    // Error code
    nErrorId: UDINT;
    // Message associated with bError = TRUE
    sErrorMessage: STRING;
    // If TRUE, we are currently moving between states
    bBusy: BOOL;
    // If TRUE, we asked for a move between states, it completed successfully, and there is no ongoing move
    bDone: BOOL;
    // The current state readback
    {attribute 'pytmc' := '
        pv: GET
        io: i
    '}
    enumGet: ENUM_EpicsInOut_INT; // NOTE: Please copy this pragma exactly on your enumGet
END_VAR
VAR
    bInit: BOOL;
    arrStates: ARRAY[1..15] OF ST_PositionState;

    {attribute 'pytmc' := '
        pv:
        io: io
    '}
    fbStateManager: FB_PositionStateManager; // NOTE: Please copy this pragma exactly to pick up the standard PVs
END_VAR

// Fist cycle setup
IF NOT bInit THEN
    stOut.sName := 'OUT';
    stIn.sName := 'IN';
    bInit := TRUE;
END_IF

// Stuff first two values of the 15 element array for the manager
arrStates[1] := stOut;
arrStates[2] := stIn;

// Call the function block every cycle
fbStateManager(
    stMotionStage := stMotionStage,
    arrStates := arrStates,
    setState := enumSet,
    bEnable := bEnable,
    bError => bError,
    nErrorId => nErrorId,
    sErrorMessage => sErrorMessage,
    bBusy => bBusy,
    bDone => bDone,
    getState => enumGet); // Cannot do this assignment if enumGet has attribute strict

END_FUNCTION_BLOCK

// POUs/Motion/States/Examples/FB_PositionState1D_InOut
FUNCTION_BLOCK FB_PositionState1D_InOut
(*
    An example and usable drop-in instance for a 1D state device with just an IN and an OUT state.
*)
VAR_IN_OUT
    // Include a stage that can be passed into the FB
    stMotionStage: ST_MotionStage;
    // Simplify the interface, the user just needs to construct and pass in and out position states
    stIn: ST_PositionState;
    stOut: ST_PositionState;
END_VAR
VAR_INPUT
    // Define an ENUM for EPICS to use to set a new value. It is expected this will be written to during one cycle, so don't continually apply a value here in the PLC code.
    // It is exposed as an input so we can test it using the PLC.
    {attribute 'pytmc' := '
      pv: STATE:SET
      io: io
    '}
    eStateReq: E_EpicsInOut;
END_VAR
VAR_OUTPUT
    // Define an ENUM for EPICS to use to report the new value.
    {attribute 'pytmc' := '
      pv: STATE:GET
      io: i
    '}
    eStateGet: E_EpicsInOut;
END_VAR
VAR
    // Include the standard fb with blank pv pragma
    {attribute 'pytmc' := 'pv:'}
    fbPositionState1D: FB_PositionState1D;
    // The standard fb expects a full array of position states
    astPositionState: ARRAY[1..GeneralConstants.MAX_STATES] OF ST_PositionState;
END_VAR


// Optional: default state names
IF stIn.sName = '' THEN
    stIn.sName := 'IN';
END_IF
IF stOut.sName = '' THEN
    stOut.sName := 'OUT';
END_IF

// Assemble the states array, matching the enum values
astPositionState[E_EpicsInOut.OUT] := stOut;
astPositionState[E_EpicsInOut.IN] := stIn;

// Call the main function block, passing our motors, states, enums and an enable
fbPositionState1D(
    stMotionStage:=stMotionStage,
    astPositionState:=astPositionState,
    eEnumSet:=eStateReq,
    eEnumGet:=eStateGet,
    bEnable:=TRUE,
);

// Send updates made on the array back to the inputs (VAR_IN_OUT) for maximum clarity
stOut := astPositionState[E_EpicsInOut.OUT];
stIn := astPositionState[E_EpicsInOut.IN];

END_FUNCTION_BLOCK

// POUs/Motion/States/FB_PositionState1D
FUNCTION_BLOCK FB_PositionState1D
(*
    1-Dimensional position state function block.

    This allows the user to move a motor among some set of named state positions.

    To use a states block, you must define enums that match the state options and give them pytmc pragmas.
    See FB_PositionState1D_InOut for a simple example.
    These enums must be passed in as the eEnumSet and eEnumGet VAR_IN_OUT variables.
    The enum values must match the array indices in astPositionState.

    A move will begin when eEnumSet is set to a positive, nonzero value. eEnumSet will be reset to 0 on every cycle, allowing us
    to accept a new, possibly conflicting, move request on the next cycle to interrupt the first.

    The motor must already be set up for point-to-point motion via FB_MotionStage, etc., for this function block to work properly.

    With no PMPS handling, this FB basically just links the state names with positions in both directions for set and readback.
*)
VAR_IN_OUT
    // The motor to move.
    stMotionStage: ST_MotionStage;
    // All possible position states, including unused/invalid states.
    {attribute 'pytmc' := '
        pv: STATE
        io: io
        expand: :%.2d
    '}
    astPositionState: ARRAY[1..GeneralConstants.MAX_STATES] OF ST_PositionState;
    // Set this to a nonzero value to request a new move. It will be reset to zero every cycle. This should be hooked up to a user's EPICS enum input.
    eEnumSet: UINT;
    // The current state index, or zero if we are not at a state. This should be hooked up to a user's EPICS enum output.
    eEnumGet: UINT;
END_VAR
VAR_INPUT
    // Set this to TRUE to enable input state moves, or FALSE to disable them.
    bEnable: BOOL;
    // Normal EPICS inputs, gathered into a single struct
    {attribute 'pytmc' := 'pv: STATE'}
    stEpicsToPlc: ST_StateEpicsToPlc;
END_VAR
VAR_OUTPUT
    // Normal EPICS outputs, gathered into a single struct
    {attribute 'pytmc' := 'pv: STATE'}
    stPlcToEpics: ST_StatePlcToEpics;
END_VAR
VAR
    fbCore: FB_PositionStateND_Core;
    astMotionStageMax: ARRAY[1..MotionConstants.MAX_STATE_MOTORS] OF ST_MotionStage;
    astPositionStateMax: ARRAY[1..MotionConstants.MAX_STATE_MOTORS] OF ARRAY[1..GeneralConstants.MAX_STATES] OF ST_PositionState;
END_VAR


astMotionStageMax[1] := stMotionStage;
astPositionStateMax[1] := astPositionState;

fbCore(
    astMotionStageMax:=astMotionStageMax,
    astPositionStateMax:=astPositionStateMax,
    stEpicsToPlc:=stEpicsToPlc,
    stPlcToEpics:=stPlcToEpics,
    eEnumSet:=eEnumSet,
    eEnumGet:=eEnumGet,
    bEnable:=bEnable,
    nActiveMotorCount:=1,
);

stMotionStage := astMotionStageMax[1];
astPositionState := astPositionStateMax[1];

END_FUNCTION_BLOCK

// POUs/Motion/FB_MotionStage
FUNCTION_BLOCK FB_MotionStage
(*
    Default implementation for PLC behavior when motor IOC asks for a move
    This can be extended or replaced in your PLC project if you want
    non-default behavior to arise from the motor record processing
*)
VAR_IN_OUT
    stMotionStage: ST_MotionStage;
END_VAR
VAR
    fbDriveVirtual: FB_DriveVirtual;
    fbMotionHome: FB_MotionHoming;
    fbSaveRestore: FB_EncSaveRestore;
    fbLogError: FB_LogMotionError;
    bExecute: BOOL;
    bExecMove: BOOL;
    bExecHome: BOOL;
    bFwdHit: BOOL;
    bBwdHit: BOOL;
    ftExec: F_TRIG;
    rtExec: R_TRIG;
    rtUserExec: R_TRIG;
    rtTarget: R_TRIG;
    rtHomed: R_TRIG;
    fbSetEnables: FB_SetEnables;
    bPosGoal: BOOL;
    bNegGoal: BOOL;
    fbEncoderValue: FB_EncoderValue;
    fbNCParams: FB_MotionStageNCParams;
    bNewMoveReq: BOOL;
    bPrepareDisable: BOOL;
    bMoveCmd: BOOL;
    rtMoveCmdShortcut: R_TRIG;
    rtHomeCmdShortcut: R_TRIG;
END_VAR

// Start with an accurate status
stMotionStage.Axis.ReadStatus();

// Check for the plc shortcut commands
// Used for testing or to circumvent motor record issues
rtMoveCmdShortcut(CLK:=stMotionStage.bMoveCmd);
rtHomeCmdShortcut(CLK:=stMotionStage.bHomeCmd);
// Execute on rising edge
IF rtMoveCmdShortcut.Q AND NOT stMotionStage.bExecute THEN
    stMotionStage.bExecute := TRUE;
    stMotionStage.nCommand := E_EpicsMotorCmd.MOVE_ABSOLUTE;
ELSIF rtHomeCmdShortcut.Q AND NOT stMotionStage.bExecute THEN
    stMotionStage.bExecute := TRUE;
    stMotionStage.nCommand := E_EpicsMotorCmd.HOME;
END_IF
// Always reset, even if not rising edge, so command can be issued again
IF stMotionStage.bMoveCmd OR stMotionStage.bHomeCmd THEN
    stMotionStage.bMoveCmd := FALSE;
    stMotionStage.bHomeCmd := FALSE;
END_IF

// Automatically fill the correct nCmdData for homing
IF stMotionStage.nCommand = E_EpicsMotorCmd.HOME THEN
    stMotionStage.nCmdData := stMotionStage.nHomingMode;
END_IF

// Check if the command wants to cause a move
bMoveCmd R= stMotionStage.nCmdData = E_EpicsHomeCmd.ABSOLUTE_SET;
bMoveCmd R= stMotionStage.nCmdData = E_EpicsHomeCmd.NONE;
bMoveCmd S= stMotionStage.nCommand <> E_EpicsMotorCmd.HOME;

// Handle main execs
rtUserExec(CLK := stMotionStage.bExecute);
bNewMoveReq S= rtUserExec.Q AND bMoveCmd;
bNewMoveReq R= NOT stMotionStage.bExecute;
bPrepareDisable R= bNewMoveReq;

bPosGoal := stMotionStage.stAxisStatus.fActPosition < stMotionStage.fPosition;
bNegGoal := stMotionStage.stAxisStatus.fActPosition > stMotionStage.fPosition;

// Moves are automatically allowed if no safety hooks. Otherwise, some other code will set this.
stMotionStage.bSafetyReady S= stMotionStage.bPowerSelf;

// Handle auto-enable timing
CASE stMotionStage.nEnableMode OF
    E_StageEnableMode.ALWAYS:
        stMotionStage.bEnable := TRUE;
    E_StageEnableMode.DURING_MOTION:
        IF bNewMoveReq THEN
            IF stMotionStage.nCommand = E_EpicsMotorCmd.HOME THEN
                stMotionStage.bEnable := stMotionStage.bSafetyReady;
            ELSIF bPosGoal THEN
                IF stMotionStage.bAllForwardEnable THEN
                    stMotionStage.bEnable S= stMotionStage.bSafetyReady;
                ELSIF NOT stMotionStage.bError THEN
                    // Not an error, just a warning
                    stMotionStage.sErrorMessage := 'Cannot move past positive limit.';
                    stMotionStage.bExecute := FALSE;
                END_IF
            ELSIF bNegGoal THEN
                IF stMotionStage.bAllBackwardEnable THEN
                    stMotionStage.bEnable S= stMotionStage.bSafetyReady;
                ELSIF NOT stMotionStage.bError THEN
                    // Not an error, just a warning
                    stMotionStage.sErrorMessage := 'Cannot move past negative limit.';
                    stMotionStage.bExecute := FALSE;
                END_IF
            ELSE
                // Super rare condition where we asked for a move to exactly the same floating point we're already at
                stMotionStage.bEnable S= stMotionStage.bSafetyReady;
            END_IF
            IF stMotionStage.bEnable OR stMotionStage.bError THEN
                bNewMoveReq := FALSE;
            END_IF
        END_IF
END_CASE

// Update all enable booleans
fbSetEnables(stMotionStage:=stMotionStage);

IF stMotionStage.stAxisStatus.bBusy AND NOT bExecute THEN
    // Wait for the previous move to end
    bExecute := FALSE;
ELSIF bMoveCmd THEN
    // Do not start the move until we have power and the safety system says it is OK
    bExecute := stMotionStage.bExecute AND stMotionStage.bAllEnable AND stMotionStage.bEnableDone AND stMotionStage.bSafetyReady;
ELSE
    bExecute := stMotionStage.bExecute;
END_IF

IF bExecute AND NOT stMotionStage.bError THEN
    // Reset local warnings if things are going well
    stMotionStage.sErrorMessage := '';
END_IF

// No moves allowed in error states
IF stMotionStage.bError THEN
    bExecute := FALSE;
END_IF


bExecHome := bExecute AND stMotionStage.nCommand = 10;
bExecMove := bExecute AND NOT bExecHome;

// Handle standard commands using ESS's FB
fbDriveVirtual(En:=TRUE,
    bEnable:=stMotionStage.bAllEnable,
    bReset:=stMotionStage.bReset,
    bExecute:=bExecMove,
    nCommand:=INT_TO_UINT(stMotionStage.nCommand),
    nCmdData:=INT_TO_UINT(stMotionStage.nCmdData),
    fVelocity:=stMotionStage.fVelocity,
    fPosition:=stMotionStage.fPosition,
    fAcceleration:=stMotionStage.fAcceleration,
    fDeceleration:=stMotionStage.fDeceleration,
    bLimitFwd:=stMotionStage.bAllForwardEnable,
    bLimitBwd:=stMotionStage.bAllBackwardEnable,
    bHomeSensor:=stMotionStage.bHome,
    fHomePosition:=stMotionStage.fHomePosition,
    bPowerSelf:=stMotionStage.bPowerSelf,
    nMotionAxisID=>stMotionStage.nMotionAxisID,
    Axis:=stMotionStage.Axis);

// Some custom home handling
fbMotionHome(
    stMotionStage:=stMotionStage,
    bExecute:=bExecHome);

// Update status again after the move starts or stops
stMotionStage.Axis.ReadStatus();

// Check for a new error
IF NOT stMotionStage.bError THEN
    stMotionStage.bError := fbDriveVirtual.bError;
    stMotionStage.nErrorId := fbDriveVirtual.nErrorId;
END_IF
IF NOT stMotionStage.bError THEN
    stMotionStage.bError := fbMotionHome.bError;
    stMotionStage.nErrorId := fbMotionHome.nErrorId;
END_IF
IF NOT stMotionStage.bError AND stMotionStage.bExecute AND NOT stMotionStage.bUserEnable THEN
    stMotionStage.bError := TRUE;
    stMotionStage.nErrorId := 1;
    stMotionStage.sCustomErrorMessage := 'Move requested, but user enable is disabled!';
END_IF

// Set the error message if we have one
IF stMotionStage.bError THEN
    // Hook if other code wants to inject a non-NC error
    IF stMotionStage.sCustomErrorMessage <> '' THEN
        stMotionStage.sErrorMessage := stMotionSTage.sCustomErrorMessage;
    ELSE
        stMotionStage.sErrorMessage := F_MotionErrorCodeLookup(nErrorId := stMotionStage.nErrorId);
    END_IF
END_IF

fbLogError(
    stMotionStage:=stMotionStage,
    bEnable:=TRUE);

// When we start, set the busy/done appropriately
rtExec(CLK:=bExecute);
IF rtExec.Q THEN
    stMotionStage.bBusy := TRUE;
    stMotionStage.bDone := FALSE;
END_IF

// Force everything off in case of error
IF stMotionStage.bError THEN
    stMotionStage.bBusy := FALSE;
    stMotionStage.bDone := FALSE;
    stMotionStage.bEnable := FALSE;
END_IF

// Check the limits and cancel execution if appropriate. Without this block we have infinite error spam
bFwdHit := stMotionStage.Axis.Status.PositiveDirection AND NOT stMotionStage.bAllForwardEnable;
bBwdHit := stMotionStage.Axis.Status.NegativeDirection AND NOT stMotionStage.bAllBackwardEnable;
IF (bFwdHit OR bBwdHit) AND NOT fbMotionHome.bBusy THEN
    stMotionStage.bExecute := FALSE;
END_IF

// Check done moving via user stop, fbDriveVirtual and Target Position Monitoring, or from homing.
ftExec(CLK:=stMotionStage.bExecute);
rtTarget(CLK:=(stMotionStage.Axis.Status.InTargetPosition AND fbDriveVirtual.bDone AND bExecMove));
rtHomed(CLK:=fbMotionHome.bDone AND bExecHome);
IF ftExec.Q OR rtTarget.Q OR rtHomed.Q THEN
    IF NOT stMotionStage.bDone THEN
        stMotionStage.bDone := TRUE;
        stMotionStage.bBusy := FALSE;
        IF NOT stMotionStage.Axis.Status.Error THEN
            bExecute := FALSE;
            stMotionStage.bExecute := FALSE;
        END_IF
    END_IF
END_IF

// Handle auto-disable timing
bPrepareDisable S= stMotionStage.nEnableMode = E_StageEnableMode.DURING_MOTION AND ftExec.Q;
// Delay the disable until we reach standstill, else brake issues or other race conditions
IF bPrepareDisable AND stMotionStage.Axis.Status.MotionState = MC_AXISSTATE_STANDSTILL THEN
    bPrepareDisable := FALSE;
    stMotionStage.bEnable := FALSE;
END_IF

// Get a definitive bEnabled reading
CASE stMotionStage.Axis.Status.MotionState OF
    // We are not enabled if there is an issue
    MC_AXISSTATE_UNDEFINED, MC_AXISSTATE_DISABLED, MC_AXISSTATE_ERRORSTOP:
        stMotionStage.bEnableDone := FALSE;
    ELSE
        stMotionStage.bEnableDone := TRUE;
END_CASE

// Handle the brake. TRUE means brake disabled/released
IF stMotionStage.nBrakeMode <> E_StageBrakeMode.NO_BRAKE THEN
    CASE stMotionStage.Axis.Status.MotionState OF
        MC_AXISSTATE_UNDEFINED,
        MC_AXISSTATE_DISABLED,
        MC_AXISSTATE_ERRORSTOP:
            stMotionStage.bBrakeRelease := FALSE;
        MC_AXISSTATE_STANDSTILL:
            IF stMotionStage.nBrakeMode = E_StageBrakeMode.IF_MOVING THEN
                stMotionStage.bBrakeRelease := FALSE;
            ELSE
                stMotionStage.bBrakeRelease := TRUE;
            END_IF
        ELSE
            stMotionStage.bBrakeRelease := TRUE;
    END_CASE
END_IF

// Sync the epics status struct
stMotionStage.stAxisStatus := fbDriveVirtual.stAxisStatus;
stMotionStage.stAxisStatus.bEnabled := stMotionStage.bEnableDone;

// Override homing status, dmov as appropriate
stMotionStage.bHomed := fbMotionHome.bDone AND NOT fbMotionHome.bError;
stMotionStage.stAxisStatus.bHomed := stMotionStage.bHomed;
stMotionStage.stAxisStatus.bExecute := bExecute;
stMotionStage.stAxisStatus.nCommand := 3; // If this is not 3, the IOC stops updating positions during homing

// Fill in auxiliary status info
stMotionStage.fPosDiff := stMotionStage.Axis.NcToPlc.PosDiff;

// Reset everything when bReset is flagged
IF stMotionStage.bReset THEN
    stMotionStage.bEnable := FALSE;
    stMotionStage.bReset := FALSE;
    stMotionStage.bExecute := FALSE;
    stMotionStage.bError := FALSE;
    stMotionStage.nErrorId := 0;
    stMotionStage.sErrorMessage := '';
    stMotionStage.sCustomErrorMessage := '';
    bExecute := FALSE;
END_IF

fbEncoderValue(stMotionStage:=stMotionStage);
fbNCParams(
    stMotionStage:=stMotionStage,
    bEnable:=TRUE,
    tRefreshDelay:=T#1s);

// Save and restore as long as not an absolute encoder
fbSaveRestore(
    stMotionStage:=stMotionStage,
    bEnable:=stMotionStage.nHomingMode <> E_EpicsHomeCmd.NONE);

END_FUNCTION_BLOCK

// POUs/Motion/Utils/F_MotionErrorCodeLookup
FUNCTION F_MotionErrorCodeLookup : STRING
VAR_INPUT
    nErrorId: UDINT;
END_VAR
VAR
    msg: STRING;
END_VAR

CASE nErrorId OF
    // Common NC errors
    16#4221: msg:='Requested set velocity is not allowed';
    16#4222: msg:='Requested set position is not allowed';
    16#4223: msg:='No enable for controller and/or feed';
    16#4225: msg:='Drive not ready during axis start';
    16#4260: msg:='Drive disabled';
    16#42A0: msg:='Coupled axis error';
    16#4357: msg:='Negative limit hit';
    16#4358: msg:='Positive limit hit';
    16#4395: msg:='Set velocity not allowed';
    16#4550: msg:='Stall: position lag monitoring error';
    16#4650: msg:='Drive hardware not ready to operate';
    16#4655: msg:='Invalid IO data';
    16#4467: msg:='Encoder error: invalid actual position data';
    16#4B07: msg:='Timeout axis function block after 6 seconds';
    16#4FFF: msg:='Unknown NC error (not in manual)';

    // Custom error definitions
    E_LCLSMotionError.ABORTED: msg:='Aborted move request with active move in progress';
    E_LCLSMotionError.UNSAFE: msg:='Position state unsafe';
    E_LCLSMotionError.INVALID: msg:='Position state invalid';
    E_LCLSMotionError.TEST: msg:='Fake testing error';

    // Fallbacks
    0: msg:='';
    ELSE
        msg:='Contact PCDS to add new message';
END_CASE
F_MotionErrorCodeLookup := msg;

END_FUNCTION

// tc_mca_std_lib/POUs/Motion/FB_DriveVirtual
///#########################################################
///Function block to run a virtual drive with Nc
///	Library:		
///	Tc2_MC2.lib
///
///	Global Variables:
///	
///	Data types:
///	
///	External functions:
///
///###########################################################
FUNCTION_BLOCK FB_DriveVirtual
VAR
	sVersion: STRING:='1.0.3';	
END_VAR
VAR_INPUT
	En: BOOL;
	bEnable: BOOL;
	bReset: BOOL;
	bExecute: BOOL;
	/////	nCommandLocal...
	/////	0 = Jog
	/////	1 = MoveVelocity
	/////	2 = MoveRelative
	/////	3 = MoveAbsolut
	/////	4 = MoveModulo
	/////	10 = Homing
	/////	20 = SuperInp >>>ToBe
	/////	30 = Gear
	nCommand: UINT;
	nCmdData: UINT;
	fVelocity: LREAL;
	fPosition: LREAL;
	fAcceleration: LREAL;
	fDeceleration: LREAL;
	bJogFwd: BOOL;
	bJogBwd: BOOL;
	bLimitFwd: BOOL;
	bLimitBwd: BOOL;	
	fOverride: LREAL := 100;
	bHomeSensor: BOOL;
	fHomePosition:LREAL;
	nHomeRevOffset: UINT;
	MasterAxis: AXIS_REF;
	bPowerSelf: BOOL;
END_VAR
VAR_OUTPUT
	EnO: BOOL;
	bEnabled: BOOL;
	bBusy: BOOL;
	bDone: BOOL;
	bError: BOOL;
	bHomed: BOOL;
	nErrorId: UDINT;
	nMotionAxisID:UDINT:=0;  //Axis id in Motion (NC)
	Status: ST_AxisStatus;
	fActVelocity: LREAL;
	fActPosition: LREAL;
	fActDiff: LREAL;
    sErrorMessage:STRING;
END_VAR
VAR_IN_OUT
	Axis: AXIS_REF;
END_VAR
VAR	
	nCommandLocal: UINT;
	nCmdDataLocal: UINT;
	bFirstScan: BOOL := TRUE;
	fbReset: MC_Reset;
	fbPower: MC_Power;
	fbHalt: MC_Halt;
	fbJog: MC_Jog;
	fbMoveVelocity: MC_MoveVelocity;
	fbMoveRelative: MC_MoveRelative;
	fbMoveAbsolute: MC_MoveAbsolute;
	fbMoveModulo: MC_MoveModulo;	
	fbHomeVirtual:FB_HomeVirtual;
	fbGearInDyn: MC_GearInDyn;
	fbGearOut: MC_GearOut;
	fbExecuteRiseEdge: R_TRIG;
	stAxisStatus: DUT_AxisStatus_v0_01;	
END_VAR

EnO:=En;

// Transfer nCommand and nCmdData to local copies at rising edge of bExecute (avoid issues if nCommand or nCmdData are changed during a command) 
fbExecuteRiseEdge(CLK:=bExecute);
IF fbExecuteRiseEdge.Q THEN
  nCmdDataLocal:=nCmdData;
  nCommandLocal:=nCommand;
END_IF

bHomed:=fbHomeVirtual.bHomed; //Add in DUT_AxisStatus later
bDone:=FALSE;

(*Reset*)
fbReset(
	Execute:=bReset AND Axis.Status.Error,
	Axis:=Axis,
	Done=> ,
	Busy=> ,
	Error=> ,
	ErrorID=> );

(*Power*)
IF bPowerSelf THEN
fbPower(
	Axis:=Axis,
	Enable:=bEnable,	
	Enable_Positive:=bEnable AND bLimitFwd,	
	Enable_Negative:=bEnable AND bLimitBwd,	
	Override:=fOverride,
	BufferMode:= ,
	Status=> ,
	Busy=> ,
	Active=> ,
	Error=> ,
	ErrorID=> );
END_IF

(*Halt*)
fbHalt(
	Execute:=NOT bExecute  AND (((fbMoveVelocity.Busy OR fbPower.Busy) AND (nCommandLocal=1)) OR (fbMoveRelative.Busy AND (nCommandLocal=2)) OR (fbMoveAbsolute.Busy AND (nCommandLocal=3)) OR (fbMoveModulo.Busy AND (nCommandLocal=4)) OR (fbHomeVirtual.bBusy AND (nCommandLocal=10))),
	Deceleration:=fDeceleration,
	Jerk:=0,
	BufferMode:= ,
	Options:= ,
	Axis:=Axis ,
	Done=> ,
	Busy=> ,
	Active=> ,
	CommandAborted=> ,
	Error=> ,
	ErrorID=> );

(*Jog (Command = 0)*)
fbJog(
	JogForward:=bJogFwd AND (nCommandLocal=0) ,
	JogBackwards:=bJogBwd AND (nCommandLocal=0) ,
	Mode:=UINT_TO_INT(nCmdDataLocal),
	Position:= ,
	Velocity:=fVelocity,
	Acceleration:=fAcceleration,
	Deceleration:=fDeceleration,
	Jerk:=0,
	Axis:=Axis,
	Done=> ,
	Busy=> ,
	Active=> ,
	CommandAborted=> ,
	Error=> ,
	ErrorID=> );

(*MoveVelocity (Command = 1)*)
fbMoveVelocity(
	Execute:=bExecute AND (nCommandLocal=1),
	Velocity:=ABS(fVelocity),
	Acceleration:=fAcceleration,
	Deceleration:=fDeceleration,
	Jerk:=0,
	Direction:=SEL(fVelocity<0, MC_Positive_Direction, MC_Negative_Direction),
	BufferMode:= ,
	Options:= ,
	Axis:=Axis,
	InVelocity=> ,
	Busy=> ,
	Active=> ,
	CommandAborted=> ,
	Error=> ,
	ErrorID=> );

(*MoveRelative (Command = 2)*)
fbMoveRelative(
	Execute:=bExecute AND (nCommandLocal=2), 
	Distance:=fPosition, 
	Velocity:=ABS(fVelocity), 
	Acceleration:=fAcceleration,
	Deceleration:=fDeceleration,
	Jerk:=0,
	BufferMode:= , 
	Options:= , 
	Axis:=Axis, 
	Done=> , 
	Busy=> , 
	Active=> , 
	CommandAborted=> , 
	Error=> , 
	ErrorID=> );
	
IF nCommandLocal=2 THEN
	bDone:=fbMoveRelative.Done;
END_IF
	
(*MoveAbsolute (Command = 3)*)
fbMoveAbsolute(
	Execute:=bExecute AND (nCommandLocal=3),
	Position:=fPosition,
	Velocity:=ABS(fVelocity),
	Acceleration:=fAcceleration,
	Deceleration:=fDeceleration,
	Jerk:=0,
	BufferMode:= ,
	Options:= ,
	Axis:=Axis,
	Done=> ,
	Busy=> ,
	Active=> ,
	CommandAborted=> ,
	Error=> ,
	ErrorID=> );

IF nCommandLocal=3 THEN
	bDone:=fbMoveAbsolute.Done;
END_IF

(*MoveModulo (Command = 4)*)
fbMoveModulo(
	Execute:=bExecute AND (nCommandLocal=4), 
	Position:=fPosition, 
	Velocity:=ABS(fVelocity), 
	Acceleration:=fAcceleration, 
	Deceleration:=fDeceleration, 
	Jerk:=0, 
	Direction:=UINT_TO_INT(nCmdDataLocal), 
	BufferMode:= , 
	Options:= , 
	Axis:=Axis, 
	Done=> , 
	Busy=> , 
	Active=> , 
	CommandAborted=> , 
	Error=> , 
	ErrorID=> );

IF nCommandLocal=4 THEN
	bDone:=fbMoveModulo.Done;
END_IF
	
(*Home (Command = 10)*)
fbHomeVirtual(	
	bExecute:= nCommandLocal=10 AND bExecute,
	fHomePosition:=fHomePosition,
	bHomeSensor:=bHomeSensor,
	bLimitBwd:=bLimitBwd,
	bLimitFwd:=bLimitFwd,
	nCmdData:=nCmdDataLocal,
	bReset:=bReset,
	nHomeRevOffset:=nHomeRevOffset,
	Axis:=Axis
	);
	
IF nCommandLocal=10 THEN
	bDone:=fbHomeVirtual.bDone;
END_IF
	
(*Gear (Command = 30)*)
fbGearInDyn(
	Enable:=bExecute  AND (nCommandLocal=30),
	GearRatio:=SEL(nCmdDataLocal>0, 1,fVelocity),
	Acceleration:=fAcceleration,
	Deceleration:=fDeceleration,
	Jerk:=0.0,
	BufferMode:= , 
	Options:= , 
	Master:=MasterAxis,
	Slave:=Axis,
	InGear=> , 
	Busy=> , 
	Active=> , 
	CommandAborted=> , 
	Error=> , 
	ErrorID=> );
	
fbGearOut(
	Execute:=NOT bExecute AND Axis.Status.NotMoving AND (nCommandLocal=30),
	Slave:=Axis,
	Error=>,
	Done=>,
	ErrorID=>);


IF nCommandLocal=30 THEN
	bDone:=Axis.Status.Coupled;
END_IF

(*Busy*)
bBusy:=Axis.Status.HasJob OR Axis.Status.HomingBusy OR fbHomeVirtual.bBusy;

(*Enabled*)
bEnabled:=fbPower.Status;

(*Error from functions and Nc*)
IF fbPower.Error AND fbPower.Active THEN
	bError:=fbPower.Enable;
	nErrorId:=fbPower.ErrorID;
ELSIF fbHalt.Error AND fbHalt.Active THEN
	bError:=fbHalt.Execute;
	nErrorId:=fbHalt.ErrorID;
ELSIF fbJog.Error AND nCommandLocal=0 (*fbJog.Active*) THEN
	bError:=fbJog.JogForward OR fbJog.JogBackwards;
	nErrorId:=fbJog.ErrorID;
ELSIF fbMoveVelocity.Error AND nCommandLocal=1(*fbMoveVelocity.Active*) THEN
	bError:=fbMoveVelocity.Execute;
	nErrorId:=fbMoveVelocity.ErrorID;
ELSIF fbMoveRelative.Error AND nCommandLocal=2 (*fbMoveRelative.Active*) THEN
	bError:=fbMoveRelative.Execute;
	nErrorId:=fbMoveRelative.ErrorID;
ELSIF fbMoveAbsolute.Error AND nCommandLocal=3 (*fbMoveAbsolute.Active*) THEN
	bError:=fbMoveAbsolute.Execute;
	nErrorId:=fbMoveAbsolute.ErrorID;
ELSIF fbMoveModulo.Error AND nCommandLocal=4 (*fbMoveModulo.Active*) THEN
	bError:=fbMoveModulo.Execute;
	nErrorId:=fbMoveModulo.ErrorID;
ELSIF fbHomeVirtual.bError AND nCommandLocal=10 (*fbHome.Active*) THEN
	bError:=fbHomeVirtual.bError;
	nErrorId:=fbHomeVirtual.nErrorID;
ELSIF fbGearInDyn.Error AND nCommandLocal=30 (*fbGearInDyn.Active*) THEN
	bError:=fbGearInDyn.Enable;
	nErrorId:=fbGearInDyn.ErrorID;
ELSIF fbGearOut.Error AND nCommandLocal=30 AND Axis.Status.Coupled THEN
	bError:=fbGearOut.Execute;
	nErrorId:=fbGearOut.ErrorID;
ELSIF Axis.Status.Error  THEN
	bError:=TRUE;
	nErrorId:=Axis.Status.ErrorID;
ELSIF fbHomeVirtual.bError THEN
	bError:=TRUE;
	nErrorId:=fbHomeVirtual.nErrorId;
ELSE
	bError:=FALSE;
	nErrorId:=0;
END_IF;

(*Converese nErrorID to string*)
sErrorMessage:=WORD_TO_HEXSTR(in:=TO_WORD(nErrorID) , iPrecision:= 4, bLoCase:=0 );

(*Status from Nc*)
Status:=Axis.Status;

(*Axis id in motion "motor"*)
nMotionAxisID:=axis.NcToPlc.AxisId;

(*Actual Velocity*)
fActVelocity:=Axis.NcToPlc.ActVelo;

(*Actual Position*)
IF Axis.Status.OpMode.Modulo THEN
	fActPosition:=Axis.NcToPlc.ModuloActPos;
ELSE
	fActPosition:=Axis.NcToPlc.ActPos;
END_IF

(*Actual Position*)
fActDiff:=Axis.NcToPlc.PosDiff;


//Status struct for EPICS communication
stAxisStatus.bEnable:=bEnable;
stAxisStatus.bEnabled:=bEnabled;
stAxisStatus.bError:=bError;
stAxisStatus.bExecute:=bExecute;
stAxisStatus.bHomeSensor:=bHomeSensor;
stAxisStatus.bJogBwd:=bJogBwd;
stAxisStatus.bJogFwd:=bJogFwd;
stAxisStatus.bLimitBwd:=bLimitBwd;
stAxisStatus.bLimitFwd:=bLimitFwd;
stAxisStatus.bReset:=bReset;
stAxisStatus.fAcceleration:=fAcceleration;
stAxisStatus.fActDiff:=fActDiff;
stAxisStatus.fActPosition:=fActPosition;
stAxisStatus.fActVelocity:=fActVelocity;
stAxisStatus.fDeceleration:=fDeceleration;
stAxisStatus.fOverride:=fOverride;
stAxisStatus.fPosition:=fPosition;
stAxisStatus.fVelocity:=fVelocity;
stAxisStatus.nCmdData:=nCmdData;  //Or nCmdDataLocal
stAxisStatus.nCommand:=nCommand;  //Or nCommandLocal
stAxisStatus.nErrorId:=nErrorId;
stAxisStatus.bBusy:=bBusy;
stAxisStatus.bHomed:=bHomed;

IF bFirstScan THEN
	bFirstScan:=FALSE;
END_IF

END_FUNCTION_BLOCK

// tc_mca_std_lib/POUs/Motion/Homing/FB_HomeVirtual
FUNCTION_BLOCK FB_HomeVirtual
VAR_INPUT
	En: BOOL;
	bReset: BOOL;
	bExecute: BOOL;
	nCmdData: UINT;
	bLimitFwd: BOOL;
	bLimitBwd: BOOL;	
	bHomeSensor: BOOL;	
	fHomePosition:LREAL;
	nHomeRevOffset: UINT;
END_VAR
VAR_IN_OUT
	Axis: AXIS_REF;
END_VAR
VAR_OUTPUT
	EnO: BOOL;	
	bBusy: BOOL;
	bDone: BOOL;
	bHomed:BOOL;
	bError: BOOL;
	nErrorId: UDINT;
END_VAR
VAR
	fbHomeToSwitch: FB_HomeToSwitch;
    fbHomeDirect: FB_HomeDirect; //Only used for direct homing (set of position)
    fbMoveVelocity:MC_MoveVelocity;
    fbHomePrepare:FB_HomePrepare;
	fbHomeFinish:FB_HomeFinish;    	    		
	fbExecuteRiseEdge: R_TRIG;
    nHomingState:INT:=0;
	bExecuteHomeToSwitch:BOOL:=FALSE;
	bExecuteMoveVelocity:BOOL:=FALSE;
	bExecutePrepare: BOOL:=FALSE;
	bExecuteFinish: BOOL:=FALSE;
	bExecuteHomeDirect: BOOL;
	nCmdDataLocal: UINT;  //Ensure that nCmdData is not changed during sequence
	bSequenceReady:BOOL:=TRUE;
	bRestoreNCDataNeeded: BOOL:=FALSE;
END_VAR

EnO:=En;

IF bReset THEN	
	bError:=FALSE;
	nErrorId:=0;
END_IF

// Reset when bExecute is low
IF NOT bExecute THEN
  nHomingState:=0;
  bSequenceReady:=TRUE;
  bExecuteHomeToSwitch:=FALSE;
  bExecuteHomeDirect:=FALSE;
  bExecuteMoveVelocity:=FALSE;
  bExecutePrepare:=FALSE;
  bExecuteFinish:=FALSE;
END_IF

//Reset at rinsing edge of bExecute
fbExecuteRiseEdge(CLK:=bExecute);
IF fbExecuteRiseEdge.Q THEN
  nCmdDataLocal:=nCmdData; //Ensure that nCmdData is not changed during sequence (nCmdData will only be read at a rising edge of bExecute)
  bSequenceReady:=FALSE;
  bExecutePrepare:=TRUE;  
  bRestoreNCDataNeeded:=FALSE;
  //Check if valid nCmdDataLocal
  CASE nCmdDataLocal OF  	
    1:
    2:
    3:
    4:
    15:
    ELSE //nCmdData not valid	
      bError:=TRUE;
      nErrorId:=16#4FFF;   
  END_CASE
END_IF

//############# Prepare for homing (Read from NC and reset homed flag)
fbHomePrepare(
  En:=En,
  bExecute:=bExecutePrepare AND NOT bError, // Not needed for sequence 15 (set position only, no movement))
  bReset:=bReset,
  Axis:=Axis,
);

//############# Homing Sequences:
CASE nCmdDataLocal OF  
	
   1: // Home to low limit switch
	   CASE nHomingState OF
		  0:
		    bHomed:=Axis.Status.Homed;
            // Wait for read of velocities from NC and reset of calibration flag
	        IF fbHomePrepare.bDone AND bExecute AND NOT bSequenceReady THEN
			  bRestoreNCDataNeeded:=TRUE;
			  IF bLimitBwd THEN
                nHomingState:=1;
              ELSE
				nHomingState:=2;  //Standing on limit switch go direct to state 2 
              END_IF                                          		  
	        END_IF
		  1: // wait for reach low limit then trigger fbHomeToSwitch
		    bHomed:=FALSE;
			bSequenceReady:=FALSE;
			fbMoveVelocity.Velocity:=ABS(fbHomePrepare.fVelocityToCam);
            fbMoveVelocity.Direction:=MC_Negative_Direction;
	        bExecuteMoveVelocity:=bExecute;  // Execute MC_MoveVelocity
		    IF NOT bLimitBwd AND NOT fbMoveVelocity.Busy AND Axis.Status.NotMoving THEN //MC_MoveVelocity.Busy goes down when ramp down initiates (not ends).
			  nHomingState:=2;
		    END_IF
		  2: // Wait for fbHomeToSwitch
		    bHomed:=FALSE;
		    bSequenceReady:=FALSE;
            bExecuteMoveVelocity:=FALSE;			
            bExecuteHomeToSwitch:=TRUE;	
            fbHomeToSwitch.nSearchDirTwoardsCam:=MC_Positive_Direction;
            fbHomeToSwitch.nSearchDirOffCam:=MC_Positive_Direction;	             
	        fbHomeToSwitch.fVelocityToCamNC:=fbHomePrepare.fVelocityToCam; // High speed
  	        fbHomeToSwitch.fVelocityFromCamNC:=fbHomePrepare.fVelocityFromCam;  // Low speed              		
		    fbHomeToSwitch.bCamSensor:=NOT bLimitBwd;            	 		    
	        IF fbHomeToSwitch.bDone THEN	          
			  nHomingState:=3;
			  bExecuteFinish:=TRUE;
			  fbHomeFinish.bSofLimEnableHigh:=fbHomePrepare.bSofLimEnableHighOriginal;
			  fbHomeFinish.bSofLimEnableLow:=fbHomePrepare.bSofLimEnableLowOriginal;
	        END_IF;	
          3: // restore softlimit enable
            bHomed:=FALSE;
		    bSequenceReady:=FALSE;            		            	
	        IF fbHomeFinish.bDone THEN
			  bRestoreNCDataNeeded:=FALSE;
	          bSequenceReady:=TRUE;
			  nHomingState:=0;
			  bHomed:=Axis.Status.Homed;
	        END_IF;	 
	   END_CASE;
	   
   2: // Home to high limit switch
	   CASE nHomingState OF
		  0:
		    bHomed:=Axis.Status.Homed;
            // Wait for read of velocities from NC and reset of calibration flag
	        IF fbHomePrepare.bDone AND bExecute AND NOT bSequenceReady THEN
			  bRestoreNCDataNeeded:=TRUE;
			  IF bLimitFwd THEN
                nHomingState:=1;
              ELSE
				nHomingState:=2;  //Standing on limit switch go direct to state 2 
              END_IF                                          		  
	        END_IF
		  1: // wait for reach low limit then trigger fbHomeToSwitch
		    bHomed:=FALSE;
			bSequenceReady:=FALSE;
			fbMoveVelocity.Velocity:=ABS(fbHomePrepare.fVelocityToCam);
            fbMoveVelocity.Direction:=MC_Positive_Direction;
	        bExecuteMoveVelocity:=bExecute;  // Execute MC_MoveVelocity
		    IF NOT bLimitFwd AND NOT fbMoveVelocity.Busy AND Axis.Status.NotMoving THEN //MC_MoveVelocity.Busy goes down when ramp down initiates (not ends).
			  nHomingState:=2;
		    END_IF
		  2: // Wait for fbHomeToSwitch
		    bHomed:=FALSE;
		    bSequenceReady:=FALSE;
            bExecuteMoveVelocity:=FALSE;			
            bExecuteHomeToSwitch:=TRUE;	
            fbHomeToSwitch.nSearchDirTwoardsCam:=MC_Negative_Direction;
            fbHomeToSwitch.nSearchDirOffCam:=MC_Negative_Direction;	             
	        fbHomeToSwitch.fVelocityToCamNC:=fbHomePrepare.fVelocityToCam; // High speed
  	        fbHomeToSwitch.fVelocityFromCamNC:=fbHomePrepare.fVelocityFromCam;  // Low speed              		
		    fbHomeToSwitch.bCamSensor:=NOT bLimitFwd;            	 		    
	        IF fbHomeToSwitch.bDone THEN	          
			  nHomingState:=3;
			  bExecuteFinish:=TRUE;
			  fbHomeFinish.bSofLimEnableHigh:=fbHomePrepare.bSofLimEnableHighOriginal;
			  fbHomeFinish.bSofLimEnableLow:=fbHomePrepare.bSofLimEnableLowOriginal;
	        END_IF;	
          3: // restore softlimit enable
            bHomed:=FALSE;
		    bSequenceReady:=FALSE;            		            	
	        IF fbHomeFinish.bDone THEN
			  bRestoreNCDataNeeded:=FALSE;
	          bSequenceReady:=TRUE;
			  nHomingState:=0;
			  bHomed:=Axis.Status.Homed;
	        END_IF;	 
	   END_CASE;
	   
   3: // Home on bHomeSensor via bLimitBwd
   	   CASE nHomingState OF
		  0:
		    bHomed:=Axis.Status.Homed;
            // Wait for read of velocities from NC and reset of calibration flag
	        IF fbHomePrepare.bDone AND bExecute AND NOT bSequenceReady THEN
			  bRestoreNCDataNeeded:=TRUE;
			  IF bLimitBwd THEN
                nHomingState:=1;
              ELSE
				nHomingState:=2;  //Standing on limit switch go direct to state 2 
              END_IF                                          		  
	        END_IF
		  1: // wait for reach low limit then trigger fbHomeToSwitch
		    bHomed:=FALSE;
			bSequenceReady:=FALSE;
			fbMoveVelocity.Velocity:=ABS(fbHomePrepare.fVelocityToCam);
            fbMoveVelocity.Direction:=MC_Negative_Direction;
	        bExecuteMoveVelocity:=bExecute;  // Execute MC_MoveVelocity
		    IF NOT bLimitBwd AND NOT fbMoveVelocity.Busy AND Axis.Status.NotMoving THEN //MC_MoveVelocity.Busy goes down when ramp down initiates (not ends).
			  nHomingState:=2;
		    END_IF
		  2: // Wait for fbHomeToSwitch
		    bHomed:=FALSE;
		    bSequenceReady:=FALSE;
            bExecuteMoveVelocity:=FALSE;			
            bExecuteHomeToSwitch:=TRUE;	
            fbHomeToSwitch.nSearchDirTwoardsCam:=MC_Positive_Direction;
            fbHomeToSwitch.nSearchDirOffCam:=MC_Positive_Direction;	             
	        fbHomeToSwitch.fVelocityToCamNC:=fbHomePrepare.fVelocityToCam; // High speed
  	        fbHomeToSwitch.fVelocityFromCamNC:=fbHomePrepare.fVelocityFromCam;  // Low speed              		
		    fbHomeToSwitch.bCamSensor:=bHomeSensor;            	 		    
	        IF fbHomeToSwitch.bDone THEN	          
			  nHomingState:=3;
			  bExecuteFinish:=TRUE;
			  fbHomeFinish.bSofLimEnableHigh:=fbHomePrepare.bSofLimEnableHighOriginal;
			  fbHomeFinish.bSofLimEnableLow:=fbHomePrepare.bSofLimEnableLowOriginal;
	        END_IF;	
          3: // restore softlimit enable
            bHomed:=FALSE;
		    bSequenceReady:=FALSE;            		            	
	        IF fbHomeFinish.bDone THEN
		      bRestoreNCDataNeeded:=FALSE;
	          bSequenceReady:=TRUE;
			  nHomingState:=0;
			  bHomed:=Axis.Status.Homed;
	        END_IF;	 
	   END_CASE;
	4:  // Home on bHomeSensor via bLimitFwd	   
	   CASE nHomingState OF
		  0:
		    bHomed:=Axis.Status.Homed;
            // Wait for read of velocities from NC and reset of calibration flag
	        IF fbHomePrepare.bDone AND bExecute AND NOT bSequenceReady THEN
			  bRestoreNCDataNeeded:=TRUE;
			  IF bLimitFwd THEN
                nHomingState:=1;
              ELSE
				nHomingState:=2;  //Standing on limit switch go direct to state 2 
              END_IF                                          		  
	        END_IF
		  1: // wait for reach low limit then trigger fbHomeToSwitch
		    bHomed:=FALSE;
			bSequenceReady:=FALSE;
			fbMoveVelocity.Velocity:=ABS(fbHomePrepare.fVelocityToCam);
            fbMoveVelocity.Direction:=MC_Positive_Direction;
	        bExecuteMoveVelocity:=bExecute;  // Execute MC_MoveVelocity
		    IF NOT bLimitFwd AND NOT fbMoveVelocity.Busy AND Axis.Status.NotMoving THEN //MC_MoveVelocity.Busy goes down when ramp down initiates (not ends).
			  nHomingState:=2;
		    END_IF
		  2: // Wait for fbHomeToSwitch
		    bHomed:=FALSE;
		    bSequenceReady:=FALSE;
            bExecuteMoveVelocity:=FALSE;			
            bExecuteHomeToSwitch:=TRUE;	
            fbHomeToSwitch.nSearchDirTwoardsCam:=MC_Negative_Direction;
            fbHomeToSwitch.nSearchDirOffCam:=MC_Negative_Direction;	             
	        fbHomeToSwitch.fVelocityToCamNC:=fbHomePrepare.fVelocityToCam; // High speed
  	        fbHomeToSwitch.fVelocityFromCamNC:=fbHomePrepare.fVelocityFromCam;  // Low speed              		
		    fbHomeToSwitch.bCamSensor:=bHomeSensor;            	 		    
	        IF fbHomeToSwitch.bDone THEN	          
			  nHomingState:=3;
			  bExecuteFinish:=TRUE;
			  fbHomeFinish.bSofLimEnableHigh:=fbHomePrepare.bSofLimEnableHighOriginal;
			  fbHomeFinish.bSofLimEnableLow:=fbHomePrepare.bSofLimEnableLowOriginal;
	        END_IF;	
          3: // Restore softlimit enable
            bHomed:=FALSE;
		    bSequenceReady:=FALSE;            		            	
	        IF fbHomeFinish.bDone THEN
			  bRestoreNCDataNeeded:=FALSE;
	          bSequenceReady:=TRUE;
			  nHomingState:=0;
			  bHomed:=Axis.Status.Homed;
	        END_IF;	 
	   END_CASE;
		  	    
   15: //Set current position (simplest homing sequence)
     bExecuteHomeDirect:=bExecute;
	 bHomed:=Axis.Status.Homed;
     IF fbHomeDirect.bDone THEN  //Homing ready				
	   bExecuteHomeDirect:=FALSE;				
       bSequenceReady:=TRUE;	
     END_IF	 
	 
ELSE
  fbHomeToSwitch.bCamSensor:=FALSE;
  bHomed:=Axis.Status.Homed;
END_CASE;

// Main homing block
fbHomeToSwitch(
	bExecute:=bExecuteHomeToSwitch AND bExecute AND NOT bError AND NOT bExecuteHomeDirect AND NOT bExecuteMoveVelocity,
 	bReset:=bReset,
	fHomePosition:=fHomePosition,
	Axis:=Axis
);

// Approach limit switch (error if MC_Home is used)
fbMoveVelocity(
    Execute:= bExecuteMoveVelocity AND bExecute AND NOT bError AND NOT bExecuteHomeToSwitch AND NOT bExecuteHomeDirect,
    Axis:=Axis
);

// No sequence, just set position value (nCmdDataLocal=15). Can not run if fbHomeToSwitch is executed
fbHomeDirect(
	bExecute:=bExecuteHomeDirect AND bExecute AND NOT bError  AND NOT bExecuteHomeToSwitch AND NOT bExecuteMoveVelocity,
 	bReset:=bReset,
	fHomePosition:=fHomePosition,
	Axis:=Axis
);

 
//############# Finish homing

IF NOT bexecute AND bRestoreNCDataNeeded THEN  //If homing is aborted restore is needed
	bExecuteFinish:=TRUE;
	IF fbHomeFinish.bDone THEN
	  bExecuteFinish:=FALSE;
      bRestoreNCDataNeeded:=FALSE;	
	END_IF
END_IF

fbHomeFinish(
  En:=En,
  bExecute:=bExecuteFinish,
  bReset:=bReset,
  Axis:=Axis,
);

// Error handling
IF NOT bError THEN
  IF fbHomeToSwitch.bError THEN 
	bError:=fbHomeToSwitch.bError;
	nErrorId:=fbHomeToSwitch.nErrorId;
  ELSIF fbHomeDirect.bError THEN
	bError:=fbHomeDirect.bError;
	nErrorId:=fbHomeDirect.nErrorId;
  ELSIF fbMoveVelocity.Error THEN
	bError:=fbMoveVelocity.Error;
	nErrorId:=fbMoveVelocity.ErrorId;    		    		
  END_IF;	
END_IF

// Done and busy bit
bDone:=bSequenceReady AND bExecute;
bBusy:=NOT bSequenceReady;	 

RETURN;

END_FUNCTION_BLOCK

// tc_mca_std_lib/POUs/Motion/Homing/FB_HomeToSwitch
FUNCTION_BLOCK FB_HomeToSwitch
VAR_INPUT
	En: BOOL;
	bReset: BOOL;
    bExecute: BOOL;	
    bCamSensor:BOOL;	
	nSearchDirTwoardsCam: MC_Direction;
	nSearchDirOffCam: MC_Direction;
	fHomePosition:LREAL;	
	fVelocityToCamNC: LREAL; //Velcoity when searching for cam
	fVelocityFromCamNC: LREAL; // Velocity after found cam (searching for next signal transition)
END_VAR
VAR_IN_OUT
	Axis: AXIS_REF;
END_VAR
VAR_OUTPUT
	EnO: BOOL;	
	bBusy: BOOL;
	bDone: BOOL;
	bHomed:BOOL;
	bError: BOOL;
	nErrorId: UDINT;
END_VAR
VAR
	fbHome: MC_Home;	
	fbWriteHomeDirCamToNC:FB_WriteParameterInNc_v1_00;
	fbWriteHomeDirSyncToNC:FB_WriteParameterInNc_v1_00;
	fbWriteHomeModeToNC:FB_WriteParameterInNc_v1_00;
	fbWriteHomeVelocitiesToNC: FB_HomeWriteNcVelocities;
	bConfigNCDone:BOOL:=FALSE;
	fbRTrigg: R_TRIG;
END_VAR

En:=EnO;
IF bReset THEN
	bConfigNCDone:=FALSE;
	bError:=FALSE;
	nErrorId:=0;
END_IF 
	
//Start preparation of NC if rising edge on bExecute
fbRTrigg(CLK:=bExecute);
IF fbRTrigg.Q THEN
	bConfigNCDone:=FALSE;
END_IF

 
fbWriteHomeDirCamToNC(
	bExecute:=bExecute AND NOT bConfigNCDone,
	nDeviceGroup:=16#5000,
	nIndexOffset:=16#101,	//Direction for Calibration Cam Search	
	nData:=BOOL_TO_DWORD(nSearchDirTwoardsCam=MC_Negative_Direction),//BOOL_TO_DWORD(NOT bSearchDirTwoardsCam),
	Axis:=Axis
);

fbWriteHomeDirSyncToNC(
	bExecute:= bExecute AND NOT bConfigNCDone,
	nDeviceGroup:=16#5000 ,
	nIndexOffset:=16#102 , //Direction for Sync Impuls Search
	nData:=BOOL_TO_DWORD(nSearchDirOffCam=MC_Negative_Direction),//BOOL_TO_DWORD(NOT bSearchDirOffCam),
	Axis:= Axis 
);

fbWriteHomeModeToNC(
	bExecute:=bExecute AND NOT bConfigNCDone,
	nDeviceGroup:=16#5000,
	nIndexOffset:=16#107,  //Reference Mode
	nData:=1,
	Axis:=axis);
	
fbWriteHomeVelocitiesToNC(
  En:=En,
  bExecute:=bExecute AND NOT bConfigNCDone,
  bReset:=bReset,
  fVelocityFromCam:=fVelocityFromCamNC,
  fVelocityToCam:=fVelocityToCamNC,
  Axis:=Axis);

fbHome.bCalibrationCam:=bCamSensor;

fbHome(
	Execute:=bExecute AND bConfigNCDone(* AND NOT bError*),
	Position:=fHomePosition,
	HomingMode:=0,
	Axis:=Axis
	);
bBusy:=(fbHome.Busy OR (NOT bConfigNCDone AND bExecute));
bDone:=fbHome.Done AND bConfigNCDone;
bHomed:=Axis.Status.Homed;

IF (NOT bConfigNCDone) AND fbWriteHomeDirCamToNC.bDone AND fbWriteHomeDirSyncToNC.bDone AND fbWriteHomeModeToNC.bDone AND fbWriteHomeVelocitiesToNC.bDone THEN
  bConfigNCDone:=TRUE;
END_IF

//For some reason MC_HOME gives an Error for one cycle of NC-Task 1 SVB (10ms default..) so filter with bExecute
bError:=(fbHome.Error AND bExecute) OR fbWriteHomeDirCamToNC.bError OR fbWriteHomeDirSyncToNC.bError OR fbWriteHomeModeToNC.bError OR fbWriteHomeVelocitiesToNC.bError;

IF (fbHome.Error AND bExecute) THEN
  nErrorId:=fbHome.ErrorID;
ELSIF fbWriteHomeDirCamToNC.bError THEN
  nErrorId:=fbWriteHomeDirCamToNC.nErrorId;
ELSIF fbWriteHomeDirSyncToNC.bError THEN
  nErrorId:=fbWriteHomeDirSyncToNC.nErrorId;
ELSIF fbWriteHomeModeToNC.bError THEN
  nErrorId:=fbWriteHomeModeToNC.nErrorId;
ELSIF fbWriteHomeVelocitiesToNC.bError THEN
  nErrorId:=fbWriteHomeVelocitiesToNC.nErrorId;  
END_IF

END_FUNCTION_BLOCK

// tc_mca_std_lib/POUs/ChangeConfig/FB_WriteParameterInNc_v1_00
///#########################################################
///Function block to write parameter in Nc.
///
///	Library:		
///	Tc2_MC2.lib
/// Tc2_System.lib
///
///	Global Variables:
///	
///	Data types:
///	
///	External functions:
///
///	History:
///	2014-02-05	v1.00	NB	Release code.
///
///	Known bugs:
///
///
///
///###########################################################
FUNCTION_BLOCK FB_WriteParameterInNc_v1_00
VAR_INPUT
	bExecute: BOOL;
	///16#4000=Axisdata, 16#5000=Encoderdata, 16#6000=Controldata, 16#7000=Drivedata
	nDeviceGroup: UDINT;
	nIndexOffset: UDINT;
	nData: DWORD;
END_VAR
VAR_OUTPUT
	bBusy: BOOL;
	bDone: BOOL;
	bError: BOOL;
	nErrorId: UDINT;
END_VAR
VAR_IN_OUT
	Axis: AXIS_REF;
END_VAR
VAR
	nState: UINT;
	fbADSWRITE: ADSWRITE;
END_VAR

(*Sequence to write parameter in Nc*)
CASE nState OF
0:  (*Start sequence. Wait until bExecute is TRUE*)
	IF bExecute THEN
		bBusy:=TRUE;
		bError:=FALSE;
		nErrorId:=0;
		nState:=10;
	END_IF

10: (*Write parameter in Nc*)
	fbADSWRITE(
		PORT:=500,
		IDXGRP:=nDeviceGroup+Axis.NcToPlc.AxisId,
		IDXOFFS:=nIndexOffset,
		LEN:=SIZEOF(nData),
		SRCADDR:=ADR(nData),
		WRITE:=TRUE);

	(*Wait until it's done or if an error occurs*)
	IF NOT fbADSWRITE.ERR THEN
		IF NOT fbADSWRITE.BUSY THEN
			fbADSWRITE(WRITE:=FALSE);
			nState:=20;
		END_IF
	ELSE
		nErrorId:=fbADSWRITE.ERRID;
		nState:=999;
	END_IF

20: (*Sequense is done. Waits until bExecute is FALSE*)
	bBusy:=FALSE;
	bDone:=TRUE;
	IF NOT bExecute THEN
		bDone:=FALSE;
		nState:=0;
	END_IF

999: (*Error in sequence*)
	bError:=TRUE;
	bBusy:=FALSE;
	bDone:=FALSE;
	fbADSWRITE(WRITE:=FALSE);
	IF NOT bExecute THEN
		nState:=0;
	END_IF

END_CASE

END_FUNCTION_BLOCK

// tc_mca_std_lib/POUs/Motion/Homing/FB_HomeWriteNcVelocities
FUNCTION_BLOCK FB_HomeWriteNcVelocities
VAR_INPUT
	En: BOOL;
	bReset: BOOL;
    bExecute: BOOL;		
	fVelocityToCam: LREAL;
	fVelocityFromCam: LREAL;	
END_VAR
VAR_IN_OUT
	Axis: AXIS_REF;
END_VAR
VAR_OUTPUT
	EnO: BOOL;	
	bBusy: BOOL;
	bDone: BOOL;
	bError: BOOL;
	nErrorId: UDINT;	
END_VAR
VAR
	fbExecuteRiseEdge: R_TRIG;
	fbWriteVelocityToCam:FB_WriteFloatParameter;
	fbWriteVelocityFromCam:FB_WriteFloatParameter;
END_VAR

En:=EnO;
IF bReset THEN
	bError:=FALSE;
	nErrorId:=0;
END_IF 

fbExecuteRiseEdge(CLK:=bExecute);

fbWriteVelocityToCam(
	bExecute:=bExecute,
	nDeviceGroup:= 16#4000,
	nIndexOffset:= 16#6,
	nData:=fVelocityToCam,
	Axis:= Axis);
	
fbWriteVelocityFromCam(
	bExecute:=bExecute,
	nDeviceGroup:= 16#4000,
	nIndexOffset:= 16#7,
	nData:=fVelocityFromCam,
	Axis:= Axis);

bBusy:=fbWriteVelocityFromCam.bBusy OR fbWriteVelocityToCam.bBusy;
bDone:=fbWriteVelocityFromCam.bDone AND fbWriteVelocityToCam.bDone AND bExecute;

bError:=fbWriteVelocityToCam.bError OR fbWriteVelocityFromCam.bError;
IF fbWriteVelocityToCam.bError THEN
  nErrorId:=fbWriteVelocityToCam.nErrorId;
ELSIF fbWriteVelocityFromCam.bError THEN
  nErrorId:=fbWriteVelocityFromCam.nErrorId;
END_IF

END_FUNCTION_BLOCK

// tc_mca_std_lib/POUs/ChangeConfig/FB_WriteFloatParameter
///#########################################################
///Function block to write parameter in Nc.
///
///	Library:		
///	Tc2_MC2.lib
/// Tc2_System.lib
///
///	Global Variables:
///	
///	Data types:
///	
///	External functions:
///
///	History:
///	2014-02-05	v1.00	NB	Release code.
///
///	Known bugs:
///
///
///
///###########################################################
FUNCTION_BLOCK FB_WriteFloatParameter
VAR_INPUT
	bExecute: BOOL;
	///16#4000=Axisdata, 16#5000=Encoderdata, 16#6000=Controldata, 16#7000=Drivedata
	nDeviceGroup: UDINT;
	nIndexOffset: UDINT;
	nData: LREAL;
END_VAR
VAR_OUTPUT
	bBusy: BOOL;
	bDone: BOOL;
	bError: BOOL;
	nErrorId: UDINT;
END_VAR
VAR_IN_OUT
	Axis: AXIS_REF;
END_VAR
VAR
	nState: UINT;
	fbADSWRITE: ADSWRITE;
END_VAR

(*Sequence to write parameter in Nc*)
CASE nState OF
0:  (*Start sequence. Wait until bExecute is TRUE*)
	IF bExecute THEN
		bBusy:=TRUE;
		bError:=FALSE;
		nErrorId:=0;
		nState:=10;
	END_IF

10: (*Write parameter in Nc*)
	fbADSWRITE(
		PORT:=500,
		IDXGRP:=nDeviceGroup+Axis.NcToPlc.AxisId,
		IDXOFFS:=nIndexOffset,
		LEN:=SIZEOF(nData),
		SRCADDR:=ADR(nData),
		WRITE:=TRUE);

	(*Wait until it's done or if an error occurs*)
	IF NOT fbADSWRITE.ERR THEN
		IF NOT fbADSWRITE.BUSY THEN
			fbADSWRITE(WRITE:=FALSE);
			nState:=20;
		END_IF
	ELSE
		nErrorId:=fbADSWRITE.ERRID;
		nState:=999;
	END_IF

20: (*Sequense is done. Waits until bExecute is FALSE*)
	bBusy:=FALSE;
	bDone:=TRUE;
	IF NOT bExecute THEN
		bDone:=FALSE;
		nState:=0;
	END_IF

999: (*Error in sequence*)
	bError:=TRUE;
	bBusy:=FALSE;
	bDone:=FALSE;
	fbADSWRITE(WRITE:=FALSE);
	IF NOT bExecute THEN
		nState:=0;
	END_IF

END_CASE

END_FUNCTION_BLOCK

// tc_mca_std_lib/POUs/Motion/Homing/FB_HomeDirect
FUNCTION_BLOCK FB_HomeDirect
VAR_INPUT
	En: BOOL;
	bReset: BOOL;
    bExecute: BOOL;	
	fHomePosition:LREAL;	
END_VAR
VAR_IN_OUT
	Axis: AXIS_REF;
END_VAR
VAR_OUTPUT
	EnO: BOOL;	
	bBusy: BOOL;
	bDone: BOOL;
	bHomed:BOOL;
	bError: BOOL;
	nErrorId: UDINT;
END_VAR
VAR
	fbHome: MC_Home;	
END_VAR

En:=EnO;
IF bReset THEN
	bError:=FALSE;
	nErrorId:=0;
END_IF 

fbHome(
	Execute:=bExecute,
	Position:=fHomePosition,
	HomingMode:=MC_Direct,
	bCalibrationCam:=FALSE,
	Axis:=Axis
	);
	
bBusy:=fbHome.Busy;
bDone:=fbHome.Done;
bHomed:=Axis.Status.Homed;

bError:=fbHome.Error; 

IF fbHome.Error THEN
  nErrorId:=fbHome.ErrorID;
END_IF

END_FUNCTION_BLOCK

// tc_mca_std_lib/POUs/Motion/Homing/FB_HomePrepare
FUNCTION_BLOCK FB_HomePrepare
VAR_INPUT
	En: BOOL;
	bReset: BOOL;
    bExecute: BOOL;	
    nCmdData: UINT;		
END_VAR
VAR_IN_OUT
	Axis: AXIS_REF;
END_VAR
VAR_OUTPUT
	EnO: BOOL;	
	bBusy: BOOL;
	bDone: BOOL;
	bError: BOOL;
	nErrorId: UDINT;
	bSofLimEnableLowOriginal: BOOL:=TRUE;
	bSofLimEnableHighOriginal: BOOL:=TRUE;	
	fVelocityToCam: LREAL:=0;
	fVelocityFromCam: LREAL:=0;		
END_VAR
VAR
	fbHomeReadSoftLimEnable:FB_HomeReadSoftLimEnable;	
	fbHomeDisableSoftLimEnable:FB_HomeWriteSoftLimEnable;
	fbHomeReadNCVelocities: FB_HomeReadNcVelocities;
	fbHomeResetCalibrationFlag:MC_Home;   //Only used for reset of calibration flag
	fbExecuteRiseEdge: R_TRIG;
	bExecuteReadNC:BOOL:=FALSE;
	bExecuteWriteNC:BOOL:=FALSE;
	nState:INT:=0;
END_VAR

En:=EnO;
IF bReset THEN
	bError:=FALSE;
	nErrorId:=0;
END_IF 

IF NOT bExecute THEN
  bExecuteReadNC:=FALSE;
  bExecuteWriteNC:=FALSE;   
  nState:=0;
END_IF

fbExecuteRiseEdge(CLK:=bExecute);
IF fbExecuteRiseEdge.Q THEN
  bExecuteReadNC:=TRUE;  
END_IF

// Read from NC
fbHomeReadNCVelocities(
  En:=En,
  bExecute:=bExecuteReadNC, // Actualy not needed for sequence 15 (set position only, no movement))
  bReset:=bReset,
  Axis:=Axis,
);

fbHomeReadSoftLimEnable(
	En:=En,
	bExecute:=bExecuteReadNC AND bExecute,
	Axis:=Axis,
	bReset:=bReset,	
);

// Reset calibration flag
fbHomeResetCalibrationFlag(
  Execute:=bExecuteReadNC,
  HomingMode:=MC_ResetCalibration,
  Axis:=Axis
);

bSofLimEnableLowOriginal:=fbHomeReadSoftLimEnable.bSofLimEnableLow;
bSofLimEnableHighOriginal:=fbHomeReadSoftLimEnable.bSofLimEnableHigh;	

fVelocityToCam:=fbHomeReadNCVelocities.fVelocityToCam;
fVelocityFromCam:=fbHomeReadNCVelocities.fVelocityFromCam;

IF bExecuteReadNC AND bExecute AND fbHomeReadSoftLimEnable.bDone THEN
	fbHomeDisableSoftLimEnable.bSofLimEnableHigh:=FALSE;
	fbHomeDisableSoftLimEnable.bSofLimEnableLow:=FALSE;
	bExecuteWriteNC:=TRUE; //Always write (only needed if enabled actually)
END_IF

// Write to NC (disable soft limits)
fbHomeDisableSoftLimEnable(
	En:=En,
	bExecute:=bExecuteWriteNC AND bExecute,
	Axis:=Axis,
	bReset:=bReset,	
);

bBusy:=fbHomeReadSoftLimEnable.bBusy OR fbHomeDisableSoftLimEnable.bBusy OR fbHomeReadNCVelocities.bBusy OR fbHomeResetCalibrationFlag.Busy;
bDone:=fbHomeReadSoftLimEnable.bDone AND fbHomeDisableSoftLimEnable.bDone AND fbHomeReadNCVelocities.bDone AND fbHomeResetCalibrationFlag.Done AND bExecute;

bError:=fbHomeReadSoftLimEnable.bError OR fbHomeDisableSoftLimEnable.bError OR fbHomeReadNCVelocities.bError OR fbHomeResetCalibrationFlag.Error;
IF fbHomeReadSoftLimEnable.bError THEN
  nErrorId:=fbHomeReadSoftLimEnable.nErrorId;
ELSIF fbHomeDisableSoftLimEnable.bError THEN
  nErrorId:=fbHomeDisableSoftLimEnable.nErrorId;
ELSIF fbHomeResetCalibrationFlag.Error THEN
  nErrorId:=fbHomeResetCalibrationFlag.ErrorId;
END_IF

END_FUNCTION_BLOCK

// tc_mca_std_lib/POUs/Motion/Homing/FB_HomeReadSoftLimEnable
FUNCTION_BLOCK FB_HomeReadSoftLimEnable
VAR_INPUT
	En: BOOL;
	bReset: BOOL;
    bExecute: BOOL;			
END_VAR
VAR_IN_OUT
	Axis: AXIS_REF;
END_VAR
VAR_OUTPUT
	EnO: BOOL;	
	bBusy: BOOL;
	bDone: BOOL;
	bError: BOOL;
	nErrorId: UDINT;	
	bSofLimEnableLow: BOOL:=TRUE;
	bSofLimEnableHigh: BOOL:=TRUE;
END_VAR
VAR
	fbReadSoftLimEnableLow:FB_ReadParameterInNc_v1_00;
	fbReadSoftLimEnableHigh:FB_ReadParameterInNc_v1_00;
END_VAR

En:=EnO;
IF bReset THEN
	bError:=FALSE;
	nErrorId:=0;
END_IF 
	
fbReadSoftLimEnableLow(
	bExecute:=bExecute,
	nDeviceGroup:= 16#5000,
	nIndexOffset:= 16#B,
	Axis:= Axis);

fbReadSoftLimEnableHigh(
	bExecute:=bExecute,
	nDeviceGroup:= 16#5000,
	nIndexOffset:= 16#C,
	Axis:= Axis);
	
bSofLimEnableLow:=DWORD_TO_BOOL(fbReadSoftLimEnableLow.nData);
bSofLimEnableHigh:=DWORD_TO_BOOL(fbReadSoftLimEnableHigh.nData);	

bBusy:=fbReadSoftLimEnableLow.bBusy OR fbReadSoftLimEnableHigh.bBusy;
bDone:=fbReadSoftLimEnableLow.bDone AND fbReadSoftLimEnableHigh.bDone AND bExecute;

bError:=fbReadSoftLimEnableLow.bError OR fbReadSoftLimEnableHigh.bError;
IF fbReadSoftLimEnableLow.bError THEN
  nErrorId:=fbReadSoftLimEnableLow.nErrorId;
ELSIF fbReadSoftLimEnableHigh.bError THEN
  nErrorId:=fbReadSoftLimEnableHigh.nErrorId;
END_IF

END_FUNCTION_BLOCK

// tc_mca_std_lib/POUs/ChangeConfig/FB_ReadParameterInNc_v1_00
///#########################################################
///Function block to read parameter in Nc.
///
///	Library:		
///	Tc2_MC2.lib
/// Tc2_System.lib
///
///	Global Variables:
///	
///	Data types:
///	
///	External functions:
///
///	History:
///	2014-02-05	v1.00	NB	Release code.
///
///	Known bugs:
///
///
///
///###########################################################
FUNCTION_BLOCK FB_ReadParameterInNc_v1_00
VAR_INPUT
	bExecute: BOOL;
	///16#4000=Axisdata, 16#5000=Encoderdata, 16#6000=Controldata, 16#7000=Drivedata
	nDeviceGroup: UDINT;
	nIndexOffset: UDINT;
END_VAR
VAR_OUTPUT
	nData: DWORD;
	bBusy: BOOL;
	bDone: BOOL;
	bError: BOOL;
	nErrorId: UDINT;
END_VAR
VAR_IN_OUT
	Axis: AXIS_REF;
END_VAR
VAR
	nState: UINT;
	fbADSREAD: ADSREAD;
END_VAR

(*Sequence to read parameter in Nc*)
CASE nState OF
0:  (*Start sequence. Wait until bExecute is TRUE*)
	IF bExecute THEN
		bBusy:=TRUE;
		bError:=FALSE;
		nErrorId:=0;
		nState:=10;
	END_IF

10: (*Read parameter in Nc*)
	fbADSREAD(
		PORT:=500,
		IDXGRP:=nDeviceGroup+Axis.NcToPlc.AxisId,
		IDXOFFS:=nIndexOffset,
		LEN:=SIZEOF(nData),
		DESTADDR:=ADR(nData),
		READ:=TRUE);

	(*Wait until it's done or if an error occurs*)
	IF NOT fbADSREAD.ERR THEN
		IF NOT fbADSREAD.BUSY THEN
			fbADSREAD(READ:=FALSE);
			nState:=20;
		END_IF
	ELSE
		nErrorId:=fbADSREAD.ERRID;
		nState:=999;
	END_IF

20: (*Sequense is done. Waits until bExecute is FALSE*)
	bBusy:=FALSE;
	bDone:=TRUE;
	IF NOT bExecute THEN
		bDone:=FALSE;
		nState:=0;
	END_IF

